	E_NORMAL_CAM_HANDLER_SEQ_STEPS.COUPLER_DETECT_IMAGE_ACQUIRE:
		gotoNextStep(gigECameraHandler.oImageAcquired, E_NORMAL_CAM_HANDLER_SEQ_STEPS.COUPLER_DETECT_IMAGE_PROCESSING);
		gotoNextStep(gigECameraHandler.oError, E_NORMAL_CAM_HANDLER_SEQ_STEPS.COUPLER_DETECT_FAILED);
	
	E_NORMAL_CAM_HANDLER_SEQ_STEPS.COUPLER_DETECT_IMAGE_PROCESSING:
		iCouplerProcessor.ic_process(iRawImage := rawImageCopy, iProcessedImage := processedImage, iDisplayableImage := displayableProcessedImage);
		gotoNextStep(iCouplerProcessor.ic_processingReady(), E_NORMAL_CAM_HANDLER_SEQ_STEPS.COUPLER_DETECT_DONE);
		gotoNextStep(iCouplerProcessor.ic_processingError(), E_NORMAL_CAM_HANDLER_SEQ_STEPS.COUPLER_DETECT_FAILED);

	E_NORMAL_CAM_HANDLER_SEQ_STEPS.COUPLER_DETECT_DONE:
		gotoNextStep(NOT iDetectCoupler, E_NORMAL_CAM_HANDLER_SEQ_STEPS.INIT);
	
	E_NORMAL_CAM_HANDLER_SEQ_STEPS.COUPLER_DETECT_FAILED:
		gotoNextStep(NOT iDetectCoupler, E_NORMAL_CAM_HANDLER_SEQ_STEPS.INIT);

// --------------------------------- MIRROR DETECT
	E_NORMAL_CAM_HANDLER_SEQ_STEPS.MIRROR_DETECT_ENABLE_LIGHT:
		gotoNextStep(isTimeExpired(T#500MS), E_NORMAL_CAM_HANDLER_SEQ_STEPS.MIRROR_DETECT_IMAGE_ACQUIRE);

	E_NORMAL_CAM_HANDLER_SEQ_STEPS.MIRROR_DETECT_IMAGE_ACQUIRE:
		gotoNextStep(gigECameraHandler.oImageAcquired, E_NORMAL_CAM_HANDLER_SEQ_STEPS.MIRROR_DETECT_IMAGE_PROCESSING);
		gotoNextStep(gigECameraHandler.oError, E_NORMAL_CAM_HANDLER_SEQ_STEPS.MIRROR_DETECT_FAILED);
	
	E_NORMAL_CAM_HANDLER_SEQ_STEPS.MIRROR_DETECT_IMAGE_PROCESSING:
		iMirrorProcessor.ic_process(iRawImage := rawImageCopy, iProcessedImage := processedImage, iDisplayableImage := displayableProcessedImage, iCameraPtr := gigECameraHandler.oCameraPtr, iCouplerCenterPoint := iCouplerProcessor.ic_getCenterPoint());
		gotoNextStep(iMirrorProcessor.ic_processingReady(), E_NORMAL_CAM_HANDLER_SEQ_STEPS.MIRROR_DETECT_DONE);
		gotoNextStep(iMirrorProcessor.ic_processingError(), E_NORMAL_CAM_HANDLER_SEQ_STEPS.MIRROR_DETECT_FAILED);

	E_NORMAL_CAM_HANDLER_SEQ_STEPS.MIRROR_DETECT_DONE:
		gotoNextStep(NOT iDetectMirror, E_NORMAL_CAM_HANDLER_SEQ_STEPS.INIT);
	
	E_NORMAL_CAM_HANDLER_SEQ_STEPS.MIRROR_DETECT_FAILED:
		gotoNextStep(NOT iDetectMirror, E_NORMAL_CAM_HANDLER_SEQ_STEPS.INIT);

ELSE
	step := E_NORMAL_CAM_HANDLER_SEQ_STEPS.INIT;
END_CASE
callMeRightAfterSwitchCase(TRUE, IING.STRING_BLANK);



gigECameraHandler(
	iDoIt := (step = E_NORMAL_CAM_HANDLER_SEQ_STEPS.UNDER_LIGHT_TEST_IMAGE_ACQUIRE),
	iReset := reset
);



oUnderlightOn := stepInBetween(E_NORMAL_CAM_HANDLER_SEQ_STEPS.UNDER_LIGHT_TEST_ENABLE_LIGHT, E_NORMAL_CAM_HANDLER_SEQ_STEPS.UNDER_LIGHT_TEST_IMAGE_PROCESSING)
	OR stepInBetween(E_NORMAL_CAM_HANDLER_SEQ_STEPS.COUPLER_DETECT_ENABLE_LIGHT, E_NORMAL_CAM_HANDLER_SEQ_STEPS.COUPLER_DETECT_IMAGE_PROCESSING);

oLaserLightOn := stepInBetween(E_NORMAL_CAM_HANDLER_SEQ_STEPS.LASER_LIGHT_TEST_ENABLE_LIGHT, E_NORMAL_CAM_HANDLER_SEQ_STEPS.LASER_LIGHT_TEST_IMAGE_PROCESSING);
//	OR 

oUnderLightTestOk := (step = E_NORMAL_CAM_HANDLER_SEQ_STEPS.UNDER_LIGHT_TEST_OK);
oUnderLightTestFailed := (step = E_NORMAL_CAM_HANDLER_SEQ_STEPS.UNDER_LIGHT_TEST_FAILED);

oLaserLightTestOk := (step = E_NORMAL_CAM_HANDLER_SEQ_STEPS.LASER_LIGHT_TEST_OK);
oLaserLightTestFailed := (step = E_NORMAL_CAM_HANDLER_SEQ_STEPS.LASER_LIGHT_TEST_FAILED);

oCouplerDetectDone := (step = E_NORMAL_CAM_HANDLER_SEQ_STEPS.COUPLER_DETECT_DONE);

oCouplerDetectFailed := (step = E_NORMAL_CAM_HANDLER_SEQ_STEPS.COUPLER_DETECT_FAILED);


mHmi();

METHOD PRIVATE mHmi
END_METHOD

METHOD PUBLIC stepAsString : T_SHORT_STR
stepAsString := TO_STRING(step);
END_METHOD

END_FUNCTION_BLOCK

// ---- POUs/HP/CURING_STATION/VISION/FB_GigECamHandler.TcPOU
FUNCTION_BLOCK FB_GigECamHandler EXTENDS FB_StepperProgram	// Wrapper/handler for gigE cameras, handles camera resetting, then images can be acquired (and converted)
VAR_INPUT
	iDoIt:						BOOL;		// 
	iDoConversion:				BOOL;
	iColorSpaceTransform:		ETcVnColorSpaceTransform;
	iReset:						BOOL;
END_VAR
VAR_OUTPUT
	oReadyForOperation:		BOOL;
	oImageAcquired:			BOOL;
	oDone:					BOOL;
	oError:					BOOL;
	
	oRawImage:				ITcVnImage;
	oConvertedImage:		ITcVnImage;
	
	oCameraPtr:				POINTER TO FB_VN_GevCameraControl;
	oScalingFactor:			LREAL;
END_VAR
VAR_IN_OUT
END_VAR
VAR
	step:					E_GIGE_CAM_HANDLER_SEQ_STEPS;
	hResult:				HRESULT;
	visionState:			ETcVnCameraState;
	visionStateError:		BOOL;
	ioCameraFb:				FB_VN_GevCameraControl;
	
	
END_VAR


visionState := ioCameraFb.GetState();
visionStateError := (visionState = TCVN_CS_ERROR);



callMeRightBeforeSwitchCase(ADR(step));
CASE step OF
	E_GIGE_CAM_HANDLER_SEQ_STEPS.INIT:
		gotoNextStep(iReset OR iDoIt AND (visionState = TCVN_CS_ERROR), E_GIGE_CAM_HANDLER_SEQ_STEPS.RESET_CAMERA);
		gotoNextStep(iReset OR iDoIt AND (visionState = TCVN_CS_INITIAL), E_GIGE_CAM_HANDLER_SEQ_STEPS.READY_FOR_OPERATION);

	E_GIGE_CAM_HANDLER_SEQ_STEPS.RESET_CAMERA:
		hResult := ioCameraFb.Reset();
		hResult := FC_GetCameraScalingFactor(iCameraPtr := oCameraPtr, iHrPrev := hResult, ioScale := oScalingFactor);
		
		gotoNextStep(hResult = S_OK, E_GIGE_CAM_HANDLER_SEQ_STEPS.READY_FOR_OPERATION);
		gotoNextStep(hResult = S_FALSE, E_GIGE_CAM_HANDLER_SEQ_STEPS.ERROR);
	
	E_GIGE_CAM_HANDLER_SEQ_STEPS.READY_FOR_OPERATION:
		gotoNextStep(iDoIt, E_GIGE_CAM_HANDLER_SEQ_STEPS.TRIGGER_CAMERA);
	
	E_GIGE_CAM_HANDLER_SEQ_STEPS.TRIGGER_CAMERA:
		hResult := ioCameraFb.TriggerImage();
		gotoNextStep(FAILED(hResult) OR visionStateError, E_GIGE_CAM_HANDLER_SEQ_STEPS.ERROR);
		gotoNextStep(SUCCEEDED(hresult) AND (visionState = TCVN_CS_STARTACQUISITION) , E_GIGE_CAM_HANDLER_SEQ_STEPS.START_ACQUISITION);
	
	E_GIGE_CAM_HANDLER_SEQ_STEPS.START_ACQUISITION:
		hResult := ioCameraFb.StartAcquisition();
		gotoNextStep(FAILED(hResult) OR visionStateError, E_GIGE_CAM_HANDLER_SEQ_STEPS.ERROR);
		gotoNextStep(SUCCEEDED(hresult) AND (visionState = TCVN_CS_ACQUIRING) , E_GIGE_CAM_HANDLER_SEQ_STEPS.ACQUIRING);
		
	E_GIGE_CAM_HANDLER_SEQ_STEPS.ACQUIRING:
		hResult := ioCameraFb.GetCurrentImageUndistorted(oRawImage);
		gotoNextStep(iDoConversion AND SUCCEEDED(hResult) AND (oRawImage <> IING.ZERO_POINTER), E_GIGE_CAM_HANDLER_SEQ_STEPS.DO_COLOR_CONVERSION);
		gotoNextStep(NOT iDoConversion AND SUCCEEDED(hResult) AND (oRawImage <> IING.ZERO_POINTER), E_GIGE_CAM_HANDLER_SEQ_STEPS.ACQUIRED);
		
		gotoNextStep(FAILED(hResult), E_GIGE_CAM_HANDLER_SEQ_STEPS.ERROR); 
			
	E_GIGE_CAM_HANDLER_SEQ_STEPS.DO_COLOR_CONVERSION:
		hResult := F_VN_ConvertColorSpace(ipSrcImage := oRawImage, ipDestImage := oConvertedImage, eTransform := iColorSpaceTransform, hrPrev:= hResult);
		gotoNextStep(SUCCEEDED(hResult), E_GIGE_CAM_HANDLER_SEQ_STEPS.ACQUIRED);
		gotoNextStep(FAILED(hResult), E_GIGE_CAM_HANDLER_SEQ_STEPS.ERROR);
	
	E_GIGE_CAM_HANDLER_SEQ_STEPS.ACQUIRED:
		gotoNextStep(NOT iDoIt, E_GIGE_CAM_HANDLER_SEQ_STEPS.INIT);
	
	
	E_GIGE_CAM_HANDLER_SEQ_STEPS.ERROR:
		gotoNextStep(iReset, E_GIGE_CAM_HANDLER_SEQ_STEPS.INIT);
		
	
	
ELSE
	step := E_GIGE_CAM_HANDLER_SEQ_STEPS.INIT;
END_CASE
callMeRightAfterSwitchCase(TRUE, IING.STRING_BLANK);

oCameraPtr := adr(ioCameraFb);


oReadyForOperation := (step = E_GIGE_CAM_HANDLER_SEQ_STEPS.READY_FOR_OPERATION);
oImageAcquired := (step = E_GIGE_CAM_HANDLER_SEQ_STEPS.ACQUIRING);
oError := (step = E_GIGE_CAM_HANDLER_SEQ_STEPS.ERROR);
oDone := (step = E_GIGE_CAM_HANDLER_SEQ_STEPS.DONE);

METHOD PRIVATE calcScaleFactor : LREAL
END_METHOD

END_FUNCTION_BLOCK

// ---- POUs/HP/CURING_STATION/VISION/Mirror/FC_GetCameraScalingFactor.TcPOU
FUNCTION FC_GetCameraScalingFactor : HRESULT
VAR_INPUT
	iCameraPtr:		POINTER TO FB_VN_GevCameraControl;
	iHrPrev:			HRESULT;
END_VAR
VAR_IN_OUT
	ioScale:		LREAL;		// Will contain the millimeters for ONE pixel = scale
END_VAR
VAR
 	cameraMatrix:				TcVnMatrix3x3_LREAL;
    distortionCoefficients:		TcVnArray8_LREAL;
    rotationMatrix:				TcVnMatrix3x3_LREAL;
    translationVector:			TcVnVector3_LREAL;
	//hResult:					HRESULT;
	singlePixelPoint1:			TcVnPoint2_REAL := [0, 0];
	singlePixelPoint2:			TcVnPoint2_REAL := [0, 1];
END_VAR
VAR CONSTANT

END_VAR

// Get camera calibration parameters
iCameraPtr^.GetCameraMatrix(aCameraMatrix := cameraMatrix);
iCameraPtr^.GetDistortionCoefficients(aDistortionCoefficients := distortionCoefficients);
iCameraPtr^.GetRotationMatrix(aRotationMatrix := rotationMatrix);
iCameraPtr^.GetTranslationVector(aTranslationVector := translationVector);

singlePixelPoint1[VISION.X_COORD] := 0;
singlePixelPoint1[VISION.Y_COORD] := 0;

singlePixelPoint2[VISION.X_COORD] := 0;
singlePixelPoint2[VISION.Y_COORD] := 1;


// We ask to give the distance of point1 to point2 = 1 pixel -> this will give us the scaling factor
FC_GetCameraScalingFactor := F_VN_ImagePointsWorldDistance( 
	aImagePoint1 :=				singlePixelPoint1,
	aImagePoint2 :=				singlePixelPoint2,
	fWorldDistance :=			ioScale,
	aCameraMatrix :=			cameraMatrix,
	aDistortionCoefficients :=	distortionCoefficients,
	aRotationMatrix :=			rotationMatrix,
	aTranslationVector :=		translationVector,
	fZ :=						0,
	hrPrev :=					iHrPrev
);

END_FUNCTION

// ---- POUs/HP/CURING_STATION/VISION/Coupler/FB_CouplerImageProcessor.TcPOU
FUNCTION_BLOCK FB_CouplerImageProcessor	EXTENDS FB_StepperProgram IMPLEMENTS I_ImageProcessor		// FB responsible for VISION program detecting the coupler
VAR
	step:						E_COUPLER_PROCESSOR_STEPS;
	hResult:					HRESULT;

	rightEdgeStartPoint:		TcVnPoint2_REAL;
	rightEdgeEndPoint:			TcVnPoint2_REAL;
	rightEdgeResultContainer:	ITcVnContainer;	

	rightEdgePoint:				TcVnPoint2_REAL;
	topEdgePoints:				ARRAY [0..5] OF TcVnPoint2_REAL;
	bottomEdgePoints:			ARRAY [0..5] OF TcVnPoint2_REAL;

	topEdgestartPoint:			TcVnPoint2_REAL;
	topEdgeEndPoint:			TcVnPoint2_REAL;
	topEdgeEdgeResultContainer:	ITcVnContainer;	

	startPoint3:				TcVnPoint2_REAL;
	endPoint3:					TcVnPoint2_REAL;
	bottomEdgeResultContainer:	ITcVnContainer;
	
	i:							ULINT;

	topEdgePointAverage:		TcVnPoint2_REAL;
	bottomEdgePointAverage:		TcVnPoint2_REAL;
	
	// Result of the vision operation
	centerpoint:				TcVnPoint2_REAL;


	// Set throug hinterfaces
	doProcessing:				BOOL;
	rawImage:					ITcVnImage;				// Not owned, do not clear
	processedImage:				ITcVnImage;				// NOT owned, DO NOT clear
	displayableProcessedImage:	ITcVnDisplayableImage;	// Not owned, do not clear
	
	// 'Constants'
	searchLines:				UDINT;
	minIntensityDiff:			REAL;
	searchToLeftXOffset:		REAL;
END_VAR
VAR_STAT PERSISTENT
	settings:	ST_COUPLER_DETECT_SETTINGS;
END_VAR

searchLines := 5;
minIntensityDiff := 45;
searchToLeftXOffset := 40;

callMeRightBeforeSwitchCase(ADR(step));
CASE step OF
	E_COUPLER_PROCESSOR_STEPS.INIT:
		gotoNextStep(doProcessing, E_COUPLER_PROCESSOR_STEPS.LOCATE_RIGHT_EDGE);

	E_COUPLER_PROCESSOR_STEPS.LOCATE_RIGHT_EDGE:
		//mInternalCleanup();
		rightEdgeStartPoint[VISION.X_COORD] :=		1000;
		rightEdgeStartPoint[VISION.Y_COORD] :=		1000;
		rightEdgeEndPoint[VISION.X_COORD] :=		550;
		rightEdgeEndPoint[VISION.Y_COORD] :=		1000;

		hResult := F_VN_LocateEdge(
			ipSrcImage :=		rawImage, 
			ipEdgePoints :=		rightEdgeResultContainer, 
			aStartPoint :=		rightEdgeStartPoint, 
			aEndPoint :=		rightEdgeEndPoint, 
			eEdgeDirection :=	ETcVnEdgeDirection.TCVN_ED_Light_TO_Dark, 
			fMinStrength :=		minIntensityDiff, 
			nSearchLines :=		searchLines, 				// Was 5!?!?!
			hrPrev :=			hResult
		);
		// Reads the result from the container and stores to the rightEdgePoint -> Used in the next operations for calculating an offset
//		hResult := F_VN_GetAt_TcVnVector2_REAL(ipContainer := rightEdgeResultContainer, aElement := rightEdgePoint, nIndex := 0, hrPrev := hResult);		// ONLY 1 point USED!!
		hResult := FC_ExtractFromContainerAndCalculateAvg(ipContainer := rightEdgeResultContainer, iNumOfElements := (searchLines - 1), hrPrev := hResult, ioResult := rightEdgePoint);	


		gotoNextStep(SUCCEEDED(hResult), E_COUPLER_PROCESSOR_STEPS.LOCATE_TOP_EDGE);
		gotoNextStep(FAILED(hResult), E_COUPLER_PROCESSOR_STEPS.ERROR);
	
	E_COUPLER_PROCESSOR_STEPS.LOCATE_TOP_EDGE:
		topEdgestartPoint[VISION.X_COORD] :=	rightEdgePoint[VISION.X_COORD] - searchToLeftXOffset;
		topEdgestartPoint[VISION.Y_COORD] :=	600;
		topEdgeEndPoint[VISION.X_COORD] :=		rightEdgePoint[VISION.X_COORD] - searchToLeftXOffset;
		topEdgeEndPoint[VISION.Y_COORD] :=		1000;	
		
		hResult := F_VN_LocateEdge(
			ipSrcImage :=		rawImage,
			ipEdgePoints :=		topEdgeEdgeResultContainer,
			aStartPoint :=		topEdgestartPoint,
			aEndPoint :=		topEdgeEndPoint,
			eEdgeDirection :=	ETcVnEdgeDirection.TCVN_ED_Light_TO_Dark,
			fMinStrength :=		minIntensityDiff,
			nSearchLines :=		searchLines,		// Was 4!?!?!
			hrPrev :=			hResult, 
		);
		gotoNextStep(SUCCEEDED(hResult), E_COUPLER_PROCESSOR_STEPS.LOCATE_BOTTOM_EDGE);
		gotoNextStep(FAILED(hResult), E_COUPLER_PROCESSOR_STEPS.ERROR);

	E_COUPLER_PROCESSOR_STEPS.LOCATE_BOTTOM_EDGE:
		startPoint3[VISION.X_COORD] :=		rightEdgePoint[0] - searchToLeftXOffset;
		startPoint3[VISION.Y_COORD] :=		1400;
		endPoint3[VISION.X_COORD] :=		rightEdgePoint[0] - searchToLeftXOffset;
		endPoint3[VISION.Y_COORD] :=		1000;	

		hResult := F_VN_LocateEdge(
			ipSrcImage :=		rawImage,
			ipEdgePoints :=		bottomEdgeResultContainer,
			aStartPoint :=		startPoint3,
			aEndPoint :=		endPoint3,
			eEdgeDirection :=	ETcVnEdgeDirection.TCVN_ED_Light_TO_Dark,
			fMinStrength :=		minIntensityDiff,
			nSearchLines :=		searchLines,				// Was 4!?!?!
			hrPrev :=			hResult 
		);
		gotoNextStep(SUCCEEDED(hResult), E_COUPLER_PROCESSOR_STEPS.DRAW_POINTS);
		gotoNextStep(FAILED(hResult), E_COUPLER_PROCESSOR_STEPS.ERROR);

	E_COUPLER_PROCESSOR_STEPS.DRAW_POINTS:
		hResult := F_VN_DrawPoints(ipPoints := rightEdgeResultContainer, ipDestImage := processedImage, eShape := ETcVnDrawShape.TCVN_DS_X, aColor := Color.Lime, hrPrev := hResult);
		hResult := F_VN_DrawPoints(ipPoints := topEdgeEdgeResultContainer, ipDestImage := processedImage, eShape := ETcVnDrawShape.TCVN_DS_X, aColor := Color.Lime, hrPrev := hResult);
		hResult := F_VN_DrawPoints(ipPoints := bottomEdgeResultContainer, ipDestImage := processedImage, eShape := ETcVnDrawShape.TCVN_DS_X, aColor := Color.Lime, hrPrev := hResult);

		hResult := FC_ExtractFromContainerAndCalculateAvg(ipContainer := topEdgeEdgeResultContainer, iNumOfElements := (searchLines - 1), hrPrev := hResult, ioResult := topEdgePointAverage);
		hResult := FC_ExtractFromContainerAndCalculateAvg(ipContainer := bottomEdgeResultContainer, iNumOfElements := (searchLines - 1), hrPrev := hResult, ioResult := bottomEdgePointAverage);
		centerpoint := FC_CalculateCenterPoint(topEdgePointAverage, bottomEdgePointAverage);

		gotoNextStep(SUCCEEDED(hResult), E_COUPLER_PROCESSOR_STEPS.MAKE_DISPLAYABLE);
		gotoNextStep(FAILED(hResult), E_COUPLER_PROCESSOR_STEPS.ERROR);	

	E_COUPLER_PROCESSOR_STEPS.MAKE_DISPLAYABLE:
		hResult := F_VN_CopyIntoDisplayableImage(processedImage, displayableProcessedImage, hResult);
		gotoNextStep(SUCCEEDED(hResult), E_COUPLER_PROCESSOR_STEPS.DONE);
		gotoNextStep(FAILED(hResult), E_COUPLER_PROCESSOR_STEPS.ERROR);
	
	E_COUPLER_PROCESSOR_STEPS.DONE:
		gotoNextStep(NOT doProcessing, E_COUPLER_PROCESSOR_STEPS.INIT);
	
	E_COUPLER_PROCESSOR_STEPS.ERROR:
		gotoNextStep(NOT doProcessing, E_COUPLER_PROCESSOR_STEPS.INIT);
	
ELSE
	step := E_COUPLER_PROCESSOR_STEPS.INIT;
END_CASE
callMeRightAfterSwitchCase(TRUE, IING.STRING_BLANK);

METHOD PRIVATE _mInternalCleanup
doProcessing := FALSE;
END_METHOD

METHOD ic_cancelProcessing
VAR_INPUT
END_VAR
doProcessing := FALSE;
END_METHOD

METHOD ic_getCenterPoint : TcVnPoint2_REAL
ic_getCenterPoint := centerpoint;
END_METHOD

METHOD ic_process
VAR_INPUT
	iRawImage:			ITcVnImage;
	iProcessedImage:	ITcVnImage;
	iDisplayableImage:	ITcVnDisplayableImage;
END_VAR
doProcessing := TRUE;
rawImage := iRawImage;
processedImage := iProcessedImage;
displayableProcessedImage := iDisplayableImage;
END_METHOD

METHOD public ic_processingError : BOOL
ic_processingError := (step = E_COUPLER_PROCESSOR_STEPS.ERROR);
END_METHOD

METHOD public ic_processingReady : BOOL
ic_processingReady := (step = E_COUPLER_PROCESSOR_STEPS.DONE);
END_METHOD

METHOD PUBLIC stepAsString : T_SHORT_STR
stepAsString := TO_STRING(step);
END_METHOD

END_FUNCTION_BLOCK

// ---- POUs/HP/CURING_STATION/VISION/HelperFunctions/FC_ExtractFromContainerAndCalculateAvg.TcPOU
FUNCTION FC_ExtractFromContainerAndCalculateAvg  : HRESULT		// Calculates average X and Y of the search result stored in container
VAR_INPUT
	ipContainer:	ITcVnContainer;
	iNumOfElements:	UDINT;
	hrPrev	:	HRESULT;	(* HRESULT indicating the result of previous operations (If SUCCEEDED(hrPrev) equals false, no operation is executed.) *)
END_VAR
VAR_IN_OUT
	ioResult:		TcVnPoint2_REAL;
END_VAR
VAR
	i:				UDINT;
	helperPoint:			TcVnPoint2_REAL;
	hResult:		HRESULT;
END_VAR

ioResult[VISION.X_COORD] := 0;
ioResult[VISION.Y_COORD] := 0;
hResult := hrPrev;

// Fetches result and stores to element
FOR i := 0 TO (iNumOfElements - 1) DO
	hResult := F_VN_GetAt_TcVnVector2_REAL(ipContainer := ipContainer, aElement := helperPoint, nIndex := i, hrPrev := hResult);

	// Accumulate all X's and all Y's
	ioResult[VISION.X_COORD] := ioResult[VISION.X_COORD] + helperPoint[VISION.X_COORD];
	ioResult[VISION.Y_COORD] := ioResult[VISION.Y_COORD] + helperPoint[VISION.Y_COORD];
END_FOR

// Averages the X and Y's
ioResult[VISION.X_COORD] := ioResult[VISION.X_COORD] / UDINT_TO_REAL(iNumOfElements);
ioResult[VISION.Y_COORD] := ioResult[VISION.Y_COORD] / UDINT_TO_REAL(iNumOfElements);

FC_ExtractFromContainerAndCalculateAvg := hResult;

END_FUNCTION

// ---- POUs/HP/CURING_STATION/VISION/HelperFunctions/FC_CalculateCenterPoint.TcPOU
FUNCTION FC_CalculateCenterPoint : TcVnPoint2_REAL		// Calculates the center point (X and Y) of 2 points
VAR_INPUT
	iPoint1:		TcVnPoint2_REAL;
	iPoint2:		TcVnPoint2_REAL;
END_VAR

FC_CalculateCenterPoint[VISION.X_COORD] := (iPoint1[VISION.X_COORD] + iPoint2[VISION.X_COORD]) / 2;
FC_CalculateCenterPoint[VISION.Y_COORD] := (iPoint1[VISION.Y_COORD] + iPoint2[VISION.Y_COORD]) / 2;

END_FUNCTION

// ---- POUs/HP/CURING_STATION/VISION/GenericCameraHandler/FB_GenericCameraHandler.TcPOU
FUNCTION_BLOCK FB_GenericCameraHandler EXTENDS FB_StepperProgram	
VAR_INPUT
	iDoUnderLightTest:		BOOL;
	iDoLaserTest:			BOOL;
	iDetectCoupler:			BOOL;
	iDetectMirror:			BOOL;
	
	iCouplerProcessor:		I_ImageProcessor;		// FB implementing
	iMirrorProcessor:		I_ImageProcessor;
	
END_VAR
VAR_OUTPUT
	oUnderLightTestOk:			BOOL;
	oUnderLightTestFailed:		BOOL;
	oLaserLightTestOk:			BOOL;
	oLaserLightTestFailed:		BOOL;

	oCouplerDetectDone:			BOOL;
	oCouplerDetectFailed:		BOOL;

	oHmi:						ST_NORMAL_CAM_HANDLER_HMI;
	
	oUnderlightOn:				BOOL;
	oLaserLightOn:				BOOL;
END_VAR
VAR_IN_OUT
END_VAR
VAR
	step:					E_NORMAL_CAM_HANDLER_SEQ_STEPS;
	service:				ST_NORMAL_CAM_HANDLER_SERVICE;
	
	visionState:			ETcVnCameraState;
	gigECameraHandler:		FB_GigECamHandler;
	hResult:				HRESULT;
	
	rectangleArea:			TcVnRectangle_UDINT;
	rawImageCopy:			ITcVnImage;				// Image of either under light/laser
	processedImage:			ITcVnImage;
	displayableProcessedImage:	ITcVnDisplayableImage;

	averagePixelValue:		TcVnVector4_LREAL;
	
	reset:					BOOL;
	

END_VAR
VAR PERSISTENT
	settings:				ST_NORMAL_CAM_HANDLER_SETTINGS;
END_VAR

reset := iControlSignals.resetPulse;



callMeRightBeforeSwitchCase(ADR(step));
CASE step OF
	E_NORMAL_CAM_HANDLER_SEQ_STEPS.INIT:
		gotoNextStep(iDoUnderLightTest OR service.doUnderLightTest, E_NORMAL_CAM_HANDLER_SEQ_STEPS.UNDER_LIGHT_TEST_ENABLE_LIGHT);
		gotoNextStep(iDoLaserTest OR service.doLaserTest, E_NORMAL_CAM_HANDLER_SEQ_STEPS.LASER_LIGHT_TEST_ENABLE_LIGHT);
		gotoNextStep(iDetectCoupler, E_NORMAL_CAM_HANDLER_SEQ_STEPS.COUPLER_DETECT_ENABLE_LIGHT);
		gotoNextStep(iDetectMirror, E_NORMAL_CAM_HANDLER_SEQ_STEPS.MIRROR_DETECT_ENABLE_LIGHT);



// --------------------------------- COUPLER DETECT
	E_NORMAL_CAM_HANDLER_SEQ_STEPS.COUPLER_DETECT_ENABLE_LIGHT:
		gotoNextStep(isTimeExpired(T#500MS), E_NORMAL_CAM_HANDLER_SEQ_STEPS.COUPLER_DETECT_IMAGE_ACQUIRE);

	E_NORMAL_CAM_HANDLER_SEQ_STEPS.COUPLER_DETECT_IMAGE_ACQUIRE:
		gotoNextStep(gigECameraHandler.oImageAcquired, E_NORMAL_CAM_HANDLER_SEQ_STEPS.COUPLER_DETECT_IMAGE_PROCESSING);
		gotoNextStep(gigECameraHandler.oError, E_NORMAL_CAM_HANDLER_SEQ_STEPS.COUPLER_DETECT_FAILED);
	
	E_NORMAL_CAM_HANDLER_SEQ_STEPS.COUPLER_DETECT_IMAGE_PROCESSING:
		iCouplerProcessor.ic_process(iRawImage := rawImageCopy, iProcessedImage := processedImage, iDisplayableImage := displayableProcessedImage);
		gotoNextStep(iCouplerProcessor.ic_processingReady(), E_NORMAL_CAM_HANDLER_SEQ_STEPS.COUPLER_DETECT_DONE);
		gotoNextStep(iCouplerProcessor.ic_processingError(), E_NORMAL_CAM_HANDLER_SEQ_STEPS.COUPLER_DETECT_FAILED);

	E_NORMAL_CAM_HANDLER_SEQ_STEPS.COUPLER_DETECT_DONE:
		gotoNextStep(NOT iDetectCoupler, E_NORMAL_CAM_HANDLER_SEQ_STEPS.INIT);
	
	E_NORMAL_CAM_HANDLER_SEQ_STEPS.COUPLER_DETECT_FAILED:
		gotoNextStep(NOT iDetectCoupler, E_NORMAL_CAM_HANDLER_SEQ_STEPS.INIT);


ELSE
	step := E_NORMAL_CAM_HANDLER_SEQ_STEPS.INIT;
END_CASE
callMeRightAfterSwitchCase(TRUE, IING.STRING_BLANK);



gigECameraHandler(
	iDoIt := (step = E_NORMAL_CAM_HANDLER_SEQ_STEPS.UNDER_LIGHT_TEST_IMAGE_ACQUIRE),
	iReset := reset
);



oUnderlightOn := stepInBetween(E_NORMAL_CAM_HANDLER_SEQ_STEPS.UNDER_LIGHT_TEST_ENABLE_LIGHT, E_NORMAL_CAM_HANDLER_SEQ_STEPS.UNDER_LIGHT_TEST_IMAGE_PROCESSING)
	OR stepInBetween(E_NORMAL_CAM_HANDLER_SEQ_STEPS.COUPLER_DETECT_ENABLE_LIGHT, E_NORMAL_CAM_HANDLER_SEQ_STEPS.COUPLER_DETECT_IMAGE_PROCESSING);

oLaserLightOn := stepInBetween(E_NORMAL_CAM_HANDLER_SEQ_STEPS.LASER_LIGHT_TEST_ENABLE_LIGHT, E_NORMAL_CAM_HANDLER_SEQ_STEPS.LASER_LIGHT_TEST_IMAGE_PROCESSING);
//	OR 

oUnderLightTestOk := (step = E_NORMAL_CAM_HANDLER_SEQ_STEPS.UNDER_LIGHT_TEST_OK);
oUnderLightTestFailed := (step = E_NORMAL_CAM_HANDLER_SEQ_STEPS.UNDER_LIGHT_TEST_FAILED);

oLaserLightTestOk := (step = E_NORMAL_CAM_HANDLER_SEQ_STEPS.LASER_LIGHT_TEST_OK);
oLaserLightTestFailed := (step = E_NORMAL_CAM_HANDLER_SEQ_STEPS.LASER_LIGHT_TEST_FAILED);

oCouplerDetectDone := (step = E_NORMAL_CAM_HANDLER_SEQ_STEPS.COUPLER_DETECT_DONE);

oCouplerDetectFailed := (step = E_NORMAL_CAM_HANDLER_SEQ_STEPS.COUPLER_DETECT_FAILED);


mHmi();

METHOD PRIVATE mHmi
END_METHOD

METHOD PUBLIC stepAsString : T_SHORT_STR
stepAsString := TO_STRING(step);
END_METHOD

END_FUNCTION_BLOCK

// ---- POUs/HP/CURING_STATION/VISION/Mirror/FB_MirrorImageProcessor.TcPOU
FUNCTION_BLOCK FB_MirrorImageProcessor	EXTENDS FB_StepperProgram IMPLEMENTS I_MirrorImageProcessor		// FB responsible for VISION program detecting the mirror
VAR_INPUT
	iRecipes:					REFERENCE TO ST_Recipes;
END_VAR
VAR
	step:						E_MIRROR_PROCESSOR_STEPS;
	hResult:					HRESULT;
 
	cameraScale:				LREAL;		// 1 pixel in millimeters
	mirrorCenterToWeightCenterYDiffInPixels:	LREAL;
	mirrorHalfHeightInMm:			LREAL;

	upperEdgeStartPoint:		TcVnPoint2_REAL;
	upperEdgeEndPoint:			TcVnPoint2_REAL;
	upperEdgeResultContainer:	ITcVnContainer;	

	lowerEdgeStartPoint:		TcVnPoint2_REAL;
	lowerEdgeEndPoint:			TcVnPoint2_REAL;
	lowerEdgeResultContainer:	ITcVnContainer;	

	upperEdgePointAverage:		TcVnPoint2_REAL;
	lowerEdgePointAverage:		TcVnPoint2_REAL;

	mirrorCenterY:				REAL;
	// Result of the vision operation
	yOffsetInMm:					REAL;


	// Set through hinterfaces
	doProcessing:				BOOL;
	rawImage:					ITcVnImage;				// Not owned, do not clear
	processedImage:				ITcVnImage;				// NOT owned, DO NOT clear
	displayableProcessedImage:	ITcVnDisplayableImage;	// Not owned, do not clear
	
	// 'Constants'
	searchLines:				UDINT;
	minIntensityDiff:			REAL;
	verticalSearchYOffsetInPixels:		REAL;
	cameraPtr:					POINTER TO FB_VN_GevCameraControl;
	couplerCenterPoint:			TcVnPoint2_REAL;
END_VAR
VAR_STAT PERSISTENT
	settings:	ST_MIRROR_DETECT_SETTINGS;
END_VAR
VAR CONSTANT
	SINGLE_PIXEL_POINT1:	TcVnPoint2_REAL := [0, 0];
	SINGLE_PIXEL_POINT2:	TcVnPoint2_REAL := [0, 1];
END_VAR

searchLines := 1;
minIntensityDiff := 45;
verticalsearchYOffsetInPixels := 100;


callMeRightBeforeSwitchCase(ADR(step));
CASE step OF
	E_MIRROR_PROCESSOR_STEPS.INIT:
		gotoNextStep(doProcessing, E_MIRROR_PROCESSOR_STEPS.CALC_CENTER_POINT_OFFSET);

	E_MIRROR_PROCESSOR_STEPS.CALC_CENTER_POINT_OFFSET:
		hResult := FC_GetCameraScalingFactor(iCameraPtr := cameraPtr, iHrPrev := hResult, ioScale := cameraScale);

		mirrorCenterToWeightCenterYDiffInPixels := iRecipes.Station1To5.rMirrorCenterOffsetToWeightCenterY / cameraScale; // calculates the distance in px of the mirror centerpoint to weight centerpoint. Is used to determine currect positioning of the mirror 
	
		mirrorHalfHeightInMm := iRecipes.Station1To5.rMirrorDimensions[VISION.Y_COORD] / 2;				// HOX!!!!!   To be done either for 1..5 or 6..10
	
		// Detection from center to upper edge
		upperEdgeStartPoint[VISION.X_COORD] := LREAL_TO_REAL(couplerCenterPoint[VISION.X_COORD] - ((iRecipes.Station1To5.rCouplerGroveDepth) / cameraScale) + (iRecipes.Station1To5.rMirrorGripPointOffsetToEdgeX / cameraScale)) ;
		upperEdgeStartPoint[VISION.Y_COORD] := couplerCenterPoint[VISION.Y_COORD]; // Coupler centerpoint based Y Startpoint
		upperEdgeEndPoint[VISION.X_COORD] := upperEdgeStartPoint[VISION.X_COORD];	// Copy of start = thus same X
		upperEdgeEndPoint[VISION.Y_COORD] := LREAL_TO_REAL(couplerCenterpoint[VISION.Y_COORD] - ((mirrorHalfHeightInMm - iRecipes.Station1To5.rMirrorCenterOffsetToWeightCenterY) / cameraScale) - verticalSearchYOffsetInPixels);

		// Detection from center to lower edge
		lowerEdgeStartPoint[VISION.X_COORD] := LREAL_TO_REAL(couplerCenterPoint[VISION.X_COORD] - ((iRecipes.Station1To5.rCouplerGroveDepth) / cameraScale) + (iRecipes.Station1To5.rMirrorGripPointOffsetToEdgeX / cameraScale));
		lowerEdgeStartPoint[VISION.Y_COORD] := couplerCenterPoint[VISION.Y_COORD];
		lowerEdgeEndPoint[VISION.X_COORD] := lowerEdgeStartPoint[VISION.X_COORD];	// Copy of start = thus same X
		lowerEdgeEndPoint[VISION.Y_COORD] := LREAL_TO_REAL(couplerCenterpoint[VISION.Y_COORD] + ((mirrorHalfHeightInMm - iRecipes.Station1To5.rMirrorCenterOffsetToWeightCenterY) / cameraScale) + verticalSearchYOffsetInPixels);

		gotoNextStep(SUCCEEDED(hResult), E_MIRROR_PROCESSOR_STEPS.FIND_UPPER_EDGE); 
		gotoNextStep(FAILED(hResult), E_MIRROR_PROCESSOR_STEPS.ERROR); 

	E_MIRROR_PROCESSOR_STEPS.FIND_UPPER_EDGE:
		hResult := F_VN_LocateEdge(
			ipSrcImage :=			rawImage,
			ipEdgePoints :=			upperEdgeResultContainer,
			aStartPoint :=			upperEdgeStartPoint,
			aEndPoint :=			upperEdgeEndPoint,
			eEdgeDirection :=		ETcVnEdgeDirection.TCVN_ED_DARK_TO_LIGHT,
			fMinStrength :=			minIntensityDiff,
			nSearchLines :=			searchLines,
			hrPrev :=				hResult
		);
		hResult := FC_ExtractFromContainerAndCalculateAvg(ipContainer := upperEdgeResultContainer, iNumOfElements := (searchLines - 1), hrPrev := hResult, ioResult := upperEdgePointAverage);

		gotoNextStep(SUCCEEDED(hResult), E_MIRROR_PROCESSOR_STEPS.FIND_LOWER_EDGE); 
		gotoNextStep(FAILED(hResult), E_MIRROR_PROCESSOR_STEPS.ERROR); 

	E_MIRROR_PROCESSOR_STEPS.FIND_LOWER_EDGE:
		hResult := F_VN_LocateEdge(
			ipSrcImage :=			rawImage,
			ipEdgePoints :=			lowerEdgeResultContainer,
			aStartPoint :=			lowerEdgeStartPoint,
			aEndPoint :=			lowerEdgeEndPoint,
			eEdgeDirection :=		ETcVnEdgeDirection.TCVN_ED_DARK_TO_LIGHT,
			fMinStrength :=			minIntensityDiff,
			nSearchLines :=			searchLines,
			hrPrev :=				hResult
		);
		gotoNextStep(SUCCEEDED(hResult), E_MIRROR_PROCESSOR_STEPS.FIND_LOWER_EDGE); 
		gotoNextStep(FAILED(hResult), E_MIRROR_PROCESSOR_STEPS.ERROR); 

	E_MIRROR_PROCESSOR_STEPS.DRAW_POINTS:
		hResult := F_VN_DrawPoints(ipPoints := upperEdgeResultContainer, ipDestImage := processedImage, eShape := ETcVnDrawShape.TCVN_DS_X, aColor := Color.Lime, hrPrev := hResult);
		hResult := F_VN_DrawPoints(ipPoints := lowerEdgeResultContainer, ipDestImage := processedImage, eShape := ETcVnDrawShape.TCVN_DS_X, aColor := Color.Lime, hrPrev := hResult);

		// Vision found the edges of the mirror = Mirror Center
		mirrorCenterY := FC_CalculateYCenterPoint(upperEdgePointAverage, lowerEdgePointAverage);

		yOffsetInMm := LREAL_TO_REAL((couplerCenterPoint[VISION.Y_COORD] - mirrorCenterY - mirrorCenterToWeightCenterYDiffInPixels) * cameraScale);

		gotoNextStep(SUCCEEDED(hResult), E_COUPLER_PROCESSOR_STEPS.MAKE_DISPLAYABLE);
		gotoNextStep(FAILED(hResult), E_COUPLER_PROCESSOR_STEPS.ERROR);	

	E_MIRROR_PROCESSOR_STEPS.MAKE_DISPLAYABLE:
		hResult := F_VN_CopyIntoDisplayableImage(processedImage, displayableProcessedImage, hResult);
		gotoNextStep(SUCCEEDED(hResult), E_COUPLER_PROCESSOR_STEPS.DONE);
		gotoNextStep(FAILED(hResult), E_COUPLER_PROCESSOR_STEPS.ERROR);

	E_MIRROR_PROCESSOR_STEPS.DONE:
		gotoNextStep(NOT doProcessing, E_MIRROR_PROCESSOR_STEPS.INIT);
	
	E_MIRROR_PROCESSOR_STEPS.ERROR:
		gotoNextStep(NOT doProcessing, E_COUPLER_PROCESSOR_STEPS.INIT);
	
ELSE
	step := E_MIRROR_PROCESSOR_STEPS.INIT;
END_CASE
callMeRightAfterSwitchCase(TRUE, IING.STRING_BLANK);

METHOD PRIVATE _mInternalCleanup
doProcessing := FALSE;
END_METHOD

ACTION documentation:
(**









*)
END_ACTION

METHOD ic_cancelProcessing
VAR_INPUT
END_VAR
doProcessing := FALSE;
END_METHOD

METHOD ic_getResult : REAL
ic_getResult := yOffsetInMm;
END_METHOD

METHOD ic_process
VAR_INPUT
	iRawImage:				ITcVnImage;
	iProcessedImage:		ITcVnImage;
	iDisplayableImage:		ITcVnDisplayableImage;
	iCameraPtr:				POINTER TO FB_VN_GevCameraControl;
	iCouplerCenterPoint:	TcVnPoint2_REAL;					// Basis for next vision operations
END_VAR
doProcessing := TRUE;
rawImage := iRawImage;
processedImage := iProcessedImage;
displayableProcessedImage := iDisplayableImage;
cameraPtr := iCameraPtr;
couplerCenterPoint := iCouplerCenterPoint;
END_METHOD

METHOD public ic_processingError : BOOL
ic_processingError := (step = E_MIRROR_PROCESSOR_STEPS.ERROR);
END_METHOD

METHOD public ic_processingReady : BOOL
ic_processingReady := (step = E_MIRROR_PROCESSOR_STEPS.DONE);
END_METHOD

METHOD PUBLIC stepAsString : T_SHORT_STR
stepAsString := TO_STRING(step);
END_METHOD

END_FUNCTION_BLOCK

// ---- POUs/Sts/Datalog/FB_Datalogger2.TcPOU
FUNCTION_BLOCK FB_Datalogger2
VAR_INPUT
    iScaledTemp            : INT;
    stMirrorData         : REFERENCE TO ST_Vis_Mirror;
	stLaserData			: REFERENCE TO ST_Vis_Laser;
    bEnable             : BOOL;        // Rising edge = add one log entry
    bSave               : BOOL;        // Rising edge = write CSV

    Stepperpos          : LREAL;
    SensorVal           : INT;
    StepperHomed        : BOOL;
    Var4                : BOOL;
    Var5                : LREAL;
    Var6                : INT;
    Var7                : LREAL;
    Var8                : BOOL;
    Var9                : BOOL;
    Error               : BOOL;

END_VAR

VAR_OUTPUT
    bBusy               : BOOL;
    bDone               : BOOL;
    bError              : BOOL;
	bArrayWriteDone		: BOOL;
END_VAR

VAR
    // Ring buffer
    aLog        : ARRAY[0..999] OF ST_LogEntry;
    WriteIndex  : UINT := 0;
    Count       : UINT := 0;
    ReadIndex   : UINT := 0;

    // Edge detectors
    rEnable     : R_TRIG;
    rSave       : R_TRIG;

    // File handling
    fbOpen      : FB_FileOpen;
    fbWrite     : FB_FileWrite;
    fbClose     : FB_FileClose;

    hFile       : UINT;
    sLine       : STRING(255);
    sFile       : STRING(255) := 'C:\ProgramData\Beckhoff\TwinCAT\3.1\Boot\datalog2.csv';
    sCRLF       : STRING(2) := '$R$L';

    bHeaderWritten : BOOL := FALSE;
    index          : UINT;

    // State machine
    eState     : INT := 0;

    // Time stamp
    fbSysTime  : FB_LocalSystemTime;
// 					sNetID :='192.168.1.11.1.1',
// 					bEnable := TRUE);
    CurrentDT  : DT;
	
	WriteDoneTof		: TOF;
	DoneTof				: TOF;
	bDoneStatus	: BOOL;
	bWriteDone	: BOOL;
	
END_VAR

WriteDoneTof( IN := bWriteDone	, PT := T#0.2S, Q => bArrayWriteDone);
DoneTof(IN := bDoneStatus, PT := T#0.2S, Q => bDone);
bWriteDone := FALSE;
bDoneStatus := FALSE;

//  GET SYSTEM TIMESTAMP

fbSysTime(sNetID :='192.168.1.11.1.1',
					bEnable := TRUE);
//CurrentDT :=  (fbSysTime.systemTime);


//  RISING EDGE OF bEnable 

rEnable(CLK := bEnable);

IF rEnable.Q AND NOT bBusy THEN

    aLog[WriteIndex].tStamp := fbSysTime.systemTime;
    aLog[WriteIndex].Var1   := stMirrorData.rMirrorOffsetToCalPoints[1];
    aLog[WriteIndex].Var2   := stLaserData.rLaserOffsetToSetPoint[0];
    aLog[WriteIndex].Var3   := iScaledTemp;

    // Advance write pointer
    WriteIndex := WriteIndex + 1;
	bWriteDone := TRUE;
    IF WriteIndex > 999 THEN WriteIndex := 0; END_IF

    // Increment count up to 1000
    IF Count < 1000 THEN Count := Count + 1; END_IF
END_IF


//    RISING EDGE OF bSave, START FILE WRITE SEQUENCE

rSave(CLK := bSave);

IF rSave.Q AND (Count > 0) AND (NOT bBusy) THEN
    bBusy  := TRUE;
    bError := FALSE;
    eState := 10;
END_IF



CASE eState OF


// Idle

0:
    // do nothing bdone:=false????????


//  OPEN FILE (APPEND MODE)

10:
    fbOpen(
        sPathName := sFile,
        nMode     := FOPEN_MODEAPPEND,
        ePath     := PATH_GENERIC,
        bExecute  := TRUE
    );
    eState := 20;


// WAIT OPEN

20:
    fbOpen(bExecute := FALSE);

    IF NOT fbOpen.bBusy AND NOT fbOpen.bError THEN
        hFile := fbOpen.hFile;
        eState := 30;

    ELSIF fbOpen.bError THEN
        bError := TRUE;
        eState := 100;
    END_IF


// WRITE HEADER (FIRST-TIME ONLY)

30:
    IF NOT bHeaderWritten THEN
        
        sLine := 'Time,MirrorOffset,LaserOffset';
        sLine := CONCAT(sLine, sCRLF);

        fbWrite(
            hFile      := hFile,
            pWriteBuff := ADR(sLine),
            cbWriteLen := LEN(sLine),
            bExecute   := TRUE
        );

        bHeaderWritten := TRUE;
        eState := 31;

    ELSE
        ReadIndex := 0;
        eState := 40;
    END_IF


// WAIT HEADER WRITE

31:
    fbWrite(bExecute := FALSE);

    IF NOT fbWrite.bBusy AND NOT fbWrite.bError THEN
        ReadIndex := 0;
        eState := 40;
    END_IF


// WRITE LOG ENTRIES

40:
    fbWrite(bExecute := FALSE);

    IF ReadIndex < Count THEN
        
        index := (WriteIndex + 1000 - Count + ReadIndex) MOD 1000;

        // Build CSV row
        sLine := SYSTEMTIME_TO_STRING(aLog[index].tStamp);
        sLine := CONCAT(sLine, ',');
        sLine := CONCAT(sLine, LREAL_TO_STRING(aLog[index].Var1));
        sLine := CONCAT(sLine, ',');
        sLine := CONCAT(sLine, LREAL_TO_STRING(aLog[index].Var2));
        sLine := CONCAT(sLine, ',');
        sLine := CONCAT(sLine, INT_TO_STRING(aLog[index].Var3));
        sLine := CONCAT(sLine, sCRLF);

        fbWrite(
            hFile      := hFile,
            pWriteBuff := ADR(sLine),
            cbWriteLen := LEN(sLine),
            bExecute   := TRUE
        );

        eState := 41;

    ELSE
        eState := 50;
    END_IF


// WAIT LINE WRITE

41:
    fbWrite(bExecute := FALSE);

    IF NOT fbWrite.bBusy AND NOT fbWrite.bError THEN
        ReadIndex := ReadIndex + 1;
        eState := 40;   // Continue writing next entry
    END_IF


// CLOSE FILE

50:
    fbClose(hFile := hFile, bExecute := TRUE);
    eState := 60;


//WAIT CLOSE AND FINISH

60:
    fbClose(bExecute := FALSE);

    Count := 0;
    WriteIndex := 0;

    bBusy := FALSE;
    bDoneStatus := TRUE;

    eState := 0;


// ERROR

100:
    bBusy := FALSE;
    bError := TRUE;
    eState := 0;

END_CASE

END_FUNCTION_BLOCK

// ---- POUs/Sts/Datalog/FB_Datalogger3.TcPOU
FUNCTION_BLOCK FB_Datalogger3
VAR_INPUT
	iScaledTemp				: INT;
	sAssemblytype				: STRING;	//Needs to be set to the correct var in fb_stsAct, comes from st_recipe_assemblydata
	iStationIdDirect		: UDINT; // Station Id from strecipe assemblydata. 
	stMirrorData       		: REFERENCE TO ST_Vis_Mirror;
	stLaserData				: REFERENCE TO ST_Vis_Laser;
	fbHeaterControl			: REFERENCE TO FB_HeaterControl;
	stRecipeData			: reference TO ST_Recipe_AssemblyData;
                        	
    bEnable             	: BOOL;        // Rising edge = add one log entry
    bSave               	: BOOL;        // Rising edge = write CSV to a NEW timestamped file
	//istation				: INT :=8;
	stRecipeAssemblyData	: REFERENCE TO ST_Recipe_AssemblyData;
	fbStsAct				: REFERENCE TO FB_StsAct;
	
	//sMotTypeTest			: STRING := '7A6681';
//     Stepperpos          : LREAL;
//     SensorVal           : INT;
//     StepperHomed        : BOOL;
//     Var4                : BOOL;
//     Var5                : LREAL;
//     Var6                : INT;
//     Var7                : LREAL;
//     Var8                : BOOL;
//     Var9                : BOOL;
//     Error               : BOOL;
END_VAR

VAR_OUTPUT
    bBusy               	: BOOL;
    bDone               	: BOOL;
    bError              	: BOOL;
	bArrayWriteDone			: BOOL;
END_VAR                 	
                        	
VAR                     	
                        	
    aLog        			: ARRAY[0..999] OF ST_LogEntry;
    WriteIndex  			: UINT := 0;
    Count       			: UINT := 0;
    ReadIndex   			: UINT := 0;
                			
                			
    rEnable     			: R_TRIG;
    rSave       			: R_TRIG;
                			
                			
    fbOpen      			: FB_FileOpen;
    fbWrite     			: FB_FileWrite;
    fbClose     			: FB_FileClose;
                			
    hFile       			: UINT;
    sLine       			: STRING(255);
    sCRLF       			: STRING(2) := '$R$L'; // CRLF //Rivinvaihto
    // Base folder      	
    sBaseFolder 			: STRING(255) := 'C:\ProgramData\Beckhoff\TwinCAT\3.1\Boot\'; //Usbitikulle rassaus
    sFileName   			: STRING(255);		// Full path with timestamped filename
                        	
    index          			: UINT;
    eState         			: INT := 0;
                        	
                        	
    fbSysTime  				: FB_LocalSystemTime;
    CurrentDT  				: TIMESTRUCT;
                        	
                        	
    sSystemTime				: STRING(64);		//Full systemtime in string
	sTimeShort				: STRING (64);		//Shortened systemtime. Järjestelmäaika string josta millisekunnit pois
    pos        				: INT;
	iDot					: INT;				//Tunnistetaan piste sekuntien ja millis välissä
	            			
	MotorId					: STRING(64);		//Only for testing
	                    	
	WriteDoneTof			: TOF;
	DoneTof					: TOF;
	bDoneStatus				: BOOL;
	bWriteDone				: BOOL;
	
	//Station id variables
	sStationIdConvert 		: STRING;			//Asemanumeron kääntö stringiksi
	sStationID				: STRING;			//' _S'+Aseman numero stringinä
	sStationS				: STRING := '_S';	// S kirjain tiedostonimeen osoittamaan asemaa, turha? Voisi korvata '_S'
	sStationUnderScore		: STRING := '_';
	sFileNameStationId		: STRING;			// Final station id to be printed on the filename '_SX_'
	
	sFinalTimeString		: STRING;			// Aika stringinä, josta poistettu ms ja s
	SystemDT	:DT;
END_VAR

WriteDoneTof( IN := bWriteDone	, PT := T#0.2S, Q => bArrayWriteDone);
DoneTof(IN := bDoneStatus, PT := T#0.2S, Q => bDone);
bWriteDone := FALSE;
bDoneStatus := FALSE;


//Station id filename modification
sStationIDconvert := UDINT_TO_STRING (iStationIdDirect); //Käännetään asemanumero strngiksi
sStationID:=CONCAT(sStationS, sStationIDconvert); //Yhdistetään _S ja asemanumero string, syntyy _SX, jossa X asemanumero
sFileNameStationId := CONCAT (sStationID, sStationUnderScore); //Yhidstetään edellinen _SX ja alaviiva perään, syntyy _SX_


//  GET SYSTEM TIME from amsnetid
fbSysTime(sNetID :='192.168.1.11.1.1',		//192.168.1.11.1.1 //Asetettu testi-pcn amsnetid
					bEnable := TRUE);


// LOG 1 SET OF DATA WHEN bENABLE
rEnable(CLK := bEnable);

IF rEnable.Q AND NOT bBusy THEN

    aLog[WriteIndex].tStamp	:= fbSysTime.systemTime;
    aLog[WriteIndex].Var1	:= stMirrorData.rMirrorOffsetToCalPoints[1];  //stDetection.stMirror.rMirrorOffsetToCalPoints[1];
    aLog[WriteIndex].Var2	:= stLaserData.rLaserOffsetToSetPoint[0];     //stDetection.stLaser.rLaserOffsetToSetPoint[0];
    aLog[WriteIndex].Var3	:= iscaledtemp;                               //fbHeater.ScaledTemp;

    // Advance write pointer
    WriteIndex := WriteIndex + 1;
	bWriteDone := TRUE;
    IF WriteIndex > 999 THEN WriteIndex := 0; END_IF

    // Increment count to 1000
    IF Count < 1000 THEN Count := Count + 1; END_IF
END_IF



//bSave START NEW FILE WRITE 
rSave(CLK := bSave);

IF rSave.Q AND (Count > 0) AND (NOT bBusy) THEN
    
// Build filename
sSystemTime := SYSTEMTIME_TO_STRING(fbSysTime.systemTime);
//Remove millis from systemtime
iDot := FIND(sSystemTime, '.');
	IF iDot > 0 THEN
	    sTimeShort := LEFT(sSystemTime, iDot - 1);                  
	ELSE
	    sTimeShort := sSystemTime;                                   
	END_IF

// Convert : to -
FOR pos := 1 TO LEN(sTimeShort) DO
    IF sTimeShort[pos] = BYTE#58 THEN      // ':' ASCII 58
        sTimeShort[pos] := BYTE#45;        // replace with '-' ASCII 45
    END_IF
END_FOR;

// Convert  -  into _
sTimeShort[10] := BYTE#95;

sFinalTimeString := LEFT(sTimeShort, LEN(sTimeShort) - 3); //Removing seconds from the timestring

// Build final filename
sFileName := CONCAT(sBaseFolder, 'Log_');
sFileName := CONCAT(sfileName,sAssemblyType ); //Assemblynumero suoraan tähän stringinä, alaviiva logista ja asemanumerosta.
sFileName := CONCAT(sfileName,sFileNameStationId );  //Tähän viritetty station id _SX_.
sFileName := CONCAT(sFileName, sFinalTimeString); //aika ilman millis, hävitetään sekunnitkin?
sFileName := CONCAT(sFileName, '.csv');

    // Arm save sequence
    bBusy  := TRUE;
    bDone  := FALSE;
    bError := FALSE;
    eState := 10;
END_IF

//SAVE STATE MACHINE

CASE eState OF
    // Idle
    0: 
      
    // Open NEW filE
    10:
        fbOpen(
            sPathName := sFileName,
            nMode     := FOPEN_MODEWRITE,     // NEW FILE every save
            ePath     := PATH_GENERIC,
            bExecute  := TRUE
        );
        eState := 20;
    
    // Wait for file open
    20:
        fbOpen(bExecute := FALSE);

        IF NOT fbOpen.bBusy AND NOT fbOpen.bError THEN
            hFile := fbOpen.hFile;
            eState := 30;

        ELSIF fbOpen.bError THEN
            bError := TRUE;
            eState := 100;
        END_IF

    // Write header
    30:
        sLine := 'Time,MirrorOffset,LaserOffset';
        sLine := CONCAT(sLine, sCRLF);

        fbWrite(
            hFile      := hFile,
            pWriteBuff := ADR(sLine),
            cbWriteLen := LEN(sLine),
            bExecute   := TRUE
        );
        eState := 31;

    // Wait header write
    31:
        fbWrite(bExecute := FALSE);

        IF NOT fbWrite.bBusy AND NOT fbWrite.bError THEN
            ReadIndex := 0;
            eState := 40;
        END_IF

    //  Write data rows
    40:
        fbWrite(bExecute := FALSE);

        IF ReadIndex < Count THEN
            index := (WriteIndex + 1000 - Count + ReadIndex) MOD 1000; //MAKES SURE INDEX IS POSITIVE

            // Build CSV row
            sLine := SYSTEMTIME_TO_STRING(aLog[index].tStamp);  
            sLine := CONCAT(sLine, ',');
            sLine := CONCAT(sLine, LREAL_TO_STRING(aLog[index].Var1));
            sLine := CONCAT(sLine, ',');
            sLine := CONCAT(sLine, LREAL_TO_STRING(aLog[index].Var2));
            sLine := CONCAT(sLine, ',');
            sLine := CONCAT(sLine, INT_TO_STRING(aLog[index].Var3));
            sLine := CONCAT(sLine, sCRLF);

            fbWrite(
                hFile      := hFile,
                pWriteBuff := ADR(sLine),
                cbWriteLen := LEN(sLine),
                bExecute   := TRUE );

            eState := 41;

        ELSE
            eState := 50; // no more rows
        END_IF


    // Wait row write
    41:
        fbWrite(bExecute := FALSE);

        IF NOT fbWrite.bBusy AND NOT fbWrite.bError THEN
            ReadIndex := ReadIndex + 1;
            eState := 40;   // next row
        END_IF


    // Close file
    50:
        fbClose(hFile := hFile, bExecute := TRUE);
        eState := 60;

    // Finish & reset buffer
    60:
        fbClose(bExecute := FALSE);

        Count := 0;
        WriteIndex := 0;

        bBusy := FALSE;
        bDone := TRUE;
        eState := 0;
   
    100:
        bBusy := FALSE;
        bError := TRUE;
        eState := 0;

END_CASE

END_FUNCTION_BLOCK

// ---- POUs/Sts/FB_HeaterControl.TcPOU
FUNCTION_BLOCK FB_HeaterControl
VAR_INPUT
	bExecuteTest		: BOOL;
	stPlcCom			: REFERENCE TO	ST_Sts_PlcCom;
	stModulePlcCom		: REFERENCE TO ST_Module_PlcCom;
	bHeatingOnOff		: BOOL;
	bResetHeating		: BOOL;
	iStationId			: UDINT;
END_VAR
VAR_OUTPUT
	bTempReached		: BOOL := TRUE;
	bTestTempReached	: BOOL;
	ScaledTemp			: INT;
	bHeatingFailed		: BOOL;
END_VAR
VAR
	HeaterState			: INT :=0;
	HeatingTmr : TON;
	StartTmr : TON;
	iHeatingTime		: INT;
	iOffTime			: INT;
END_VAR


////////////////////////////////////////////////////////////
///////////////////////////////////////////////////////////////////
IF NOT stModulePlcCom.stPlcComIn.bEstopOk THEN
	HeaterState := 999;
	END_IF
		

ScaledTemp := (stPlcCom.stPlcComIn.PtcRawTemp / 10);

StartTmr( PT := UDINT_TO_TIME(iStationId * 2000));

IF NOT bHeatingOnOff AND NOT bExecuteTest AND stModulePlcCom.stPlcComIn.bEstopOk THEN
	HeaterState :=0;
	StartTmr.in:= FALSE;
END_IF

IF HeaterState >= 10 AND stPlcCom.stPlcComIn.PtcRawTemp >= 550 THEN
	bHeatingFailed := TRUE;
	HeaterState :=1000;
END_IF
// estoppi, jos heatingonoff false niin kaikki 0



CASE HeaterState OF
	0:	IF stModulePlcCom.stPlcComIn.bEstopOk THEN
			stPlcCom.stPlcComOut.bHeaterFan := FALSE;
			stPlcCom.stPlcComOut.bHeaterElement := FALSE;
			IF bHeatingOnOff THEN		// AND StartTmr.Q
				StartTmr.IN := TRUE;
				HeaterState := 5; //Ajastin päälle kun lämmitin tulille
			ELSIF bExecuteTest THEN
				 HeaterState := 5000;
			END_IF
		ELSE
			StartTmr.IN := FALSE;
			stPlcCom.stPlcComOut.bHeaterFan := FALSE;
			stPlcCom.stPlcComOut.bHeaterElement := FALSE;
			HeaterState := 0;	
		END_IF
		
	5:
		IF bHeatingOnOff AND StartTmr.Q THEN
			stPlcCom.stPlcComOut.bHeaterFan := TRUE;  //Ajastin päälle kun lämmitys päälle, ajastimen jälkeen lömmitin oikeasti tulille. Ajstimen nollaus kun lämmituys loppuu.
			StartTmr.IN := FALSE;
			HeaterState := 10;
		END_IF
	
	10:
		IF StPlcCom.stPlcComIn.PtcRawTemp <= 470 THEN
			iHeatingTime := 16;
			iOffTime := 4;
		ELSIF StPlcCom.stPlcComIn.PtcRawTemp <= 490 THEN
			iHeatingTime := 12;
			iOffTime := 8;
		ELSIF StPlcCom.stPlcComIn.PtcRawTemp <= 510 THEN
			iHeatingTime := 8;
			iOffTime := 12;
		ELSIF StPlcCom.stPlcComIn.PtcRawTemp <= 530 THEN
			iHeatingTime := 4;
			iOffTime := 16;
		END_IF
		HeaterState := 20;
			
	20:

		IF HeatingTmr.Q THEN
			HeatingTmr(IN:=FALSE);
			stPlcCom.stPlcComOut.bHeaterElement := FALSE;
			HeaterState := 30;
		ELSE
			HeatingTmr(IN:=TRUE,PT:=INT_TO_TIME(iHeatingTime*1000));
		END_IF
		
	30:
		IF HeatingTmr.Q THEN
			HeatingTmr(IN:=FALSE);
			stPlcCom.stPlcComOut.bHeaterElement := TRUE;
			HeaterState := 10;
		ELSE
			HeatingTmr(IN:=TRUE, PT:= INT_TO_TIME(iOffTime*1000));
		END_IF
		
	999:
		bHeatingOnOff := FALSE;
		stPlcCom.stPlcComOut.bHeaterElement := FALSE;
		stPlcCom.stPlcComOut.bHeaterFan:= FALSE;
		HeatingTmr(IN:=FALSE);
		StartTmr.IN := FALSE;
		bExecuteTest := FALSE;
			
	1000:
		bHeatingOnOff := FALSE;
		stPlcCom.stPlcComOut.bHeaterElement := FALSE;
		stPlcCom.stPlcComOut.bHeaterFan:= FALSE;
		
		IF bResetHeating THEN
			bHeatingFailed :=FALSE;
			HeaterState := 0;
		END_IF
		
//HeaterTestFunction				
	5000:
		stPlcCom.stPlcComOut.bHeaterFan := TRUE;
		IF bExecuteTest THEN
			HeaterState := 5010;
		ELSE
			HeaterState := 5000;	
		END_IF
	
	5010:
		IF stPlcCom.stPlcComIn.PtcRawTemp <= 280 THEN
				stPlcCom.stPlcComOut.bHeaterElement := TRUE;
				bTestTempReached :=FALSE;
				
			ELSIF StPlcCom.stPlcComIn.PtcRawTemp >= 280 THEN
				stPlcCom.stPlcComOut.bHeaterElement := FALSE;
				stPlcCom.stPlcComOut.bHeaterFan := FALSE;
				bTestTempReached := TRUE;
				bExecuteTest := FALSE;
				HeaterState := 5000;	
		END_IF
	
END_CASE

END_FUNCTION_BLOCK

// ---- POUs/Sts/FB_StsAct.TcPOU
FUNCTION_BLOCK FB_StsAct
VAR_IN_OUT
	bActivateStation : BOOL;
END_VAR
VAR_INPUT
	stLaserData	: REFERENCE TO ST_Vis_Laser;
	stMirrorData : REFERENCE TO ST_Vis_Mirror;
	stModuleHmi	: REFERENCE TO ST_ModuleHmi;
	stModulePlcCom	: REFERENCE TO ST_Module_PlcCom;

	bEngageSlider	:  BOOL;
	bEngageHolder : BOOL;
	bRobotReadyForStation : BOOL;
	bDismountingDone : BOOL;
	bAdjDone: BOOL;
	iStationId	: UDINT;
	rAssemblyCuringTime : REAL := 1; // IN HOURS
	bAllowStart : BOOL;
	iAdjustmentCount : INT;
	bReleaseHolders : BOOL;
END_VAR
VAR_OUTPUT
	bTrigPosCam		: BOOL;
	bTrigAngCam		: BOOL;
	bTrigPosCamLightTest	: BOOL; // triggaa testiohjelman kameralle joka katsoo että laseri, taustavalo ja itse kamera toimii. Palaute tieto on stDetectionData.stMirror.bImagingStatusOk
	bTrigPosCamLaserTest : BOOL;
	bTrigPosCamCoupler : BOOL;
	bInHoldForRobot : BOOL;
	rRobotAdjValue	: LREAL;
	bStationChecksPassed : BOOL;
	bCheckDone : BOOL;
	bHoldRobotForAdj : BOOL;
	bAssemblyFailed	: BOOL;


	sTimeLeft		: STRING;
	bDisabledByCycleDone	: BOOL;
	bPlacingDone	: BOOL;
END_VAR
VAR
	stPlcCom	: ST_Sts_PlcCom;
	fbStepper	: FB_Stepper;
	fbHeater 	: FB_HeaterControl;
	fbHeater2:	FB_CuringStationHeaterControl;
	eStationState	: E_StsActState;
	stRecipe		:ST_Recipe_AssemblyData;
	fbEventLogger		: FB_EventLogger;
	
	// PROPERTIES
	bMotorInStation	: BOOL;
	bAllPartsInStation : BOOL;
	bStationDone : BOOL;
	// MOTOR MOTION COMMANDS
	bStepForward: BOOL;
	bStepBackwards : BOOL;
	bExecuteAdj : BOOL;
	
	//INTERNAL STATUS VARIABLES
	bDetectionRetry: BOOL;
	rDetectedOffset	: LREAL;
	bLastDatalog	: BOOL;
	iStatus2Cycles	: UINT;
	bInitialStartup	: BOOL;
	bResetStation	: BOOL;
	bSetOnce : BOOL;
	bEstopCycled	: BOOL;
	iErrorId		: INT;
	sErrorId		: STRING;
	tTimeLeft		: TIME;
	iDot			: INT;
	sTime			: STRING;
	
	// CASE STEP HANDLERS
	iAssemblyCheckStep	: INT;
	iPosAdjStep			: INT;
	iStartupCheckStep	: INT;
	iStatus2Step		: INT;
	iDatalogStep		: INT;
	iMountingStep		: INT;
	
	// STATUS VARIABLES
	iAssemblyStatus : INT; // IF CURING HAS JUST BEGUN STATUS IS 1. WHEN FIRST ACCEPTED CHECK HAS OCCURED STATUS IS 2. WHEN ASSEMBLY HAS REACHED 30 MIN ACCEPETED TIME STATUS IS 3. WHEN STS IS EMPTY STATUS IS 0.
	// TIMERS
	StartupCheckTmr : TON;
	StartupStartTmr : TON;
	DataloggingTmr1 : TON;
	DataloggingTmr2	: TON;
	AssemblyDoneTmr : TON;
	bImagingTmr : TON;
	AxisResetTmr	: TON;
	MountingTmr	: TON;
	MoveTmr	: TON;
	
	fbdatalogger2		: FB_Datalogger2;
	fbdatalogger3		: FB_Datalogger3;
	
END_VAR

fbHeater(stPlcCom := stPlcCom, iStationId := iStationId, stModulePlcCom := stModulePlcCom);
fbStepper(rStepperVel := 10, stPlcCom := stPlcCom, bEstopOk := stModulePlcCom.stPlcComIn.bEstopOk);
StartupCheckTmr(PT := T#120S);
StartupStartTmr(PT := UDINT_TO_TIME(iStationId * 4 * 1000));
AssemblyDoneTmr(PT := REAL_TO_TIME(rAssemblyCuringTime * 60 * 60 * 1000));
DataloggingTmr1(PT := T#2M);
DataloggingTmr2(PT := T#5M);
bImagingTmr(PT := T#1.5S);
AxisResetTmr(PT:= T#5S);
fbdatalogger2(stMirrorData := stMirrorData, stLaserData := stLaserData, iScaledTemp := fbHeater.ScaledTemp);
fbdatalogger3(stMirrorData:=stMirrorData, stLaserData :=stLaserData, iScaledTemp := fbHeater.ScaledTemp, stRecipeAssemblyData:=stRecipe,iStationIdDirect:=iStationId, sAssemblytype:=stRecipe.sAssemblyType );
MountingTmr(PT := T#5S);
MoveTmr(PT := T#5S);
fbEventLogger(sErrorCode := sErrorId, stModuleHmi := stModuleHmi);
tTimeLeft := AssemblyDoneTmr.PT - AssemblyDoneTmr.ET;
sTime := (TIME_TO_STRING(tTimeLeft));


iDot := FIND(sTime, '.');
IF iDot > 0 THEN
	sTimeLeft := LEFT(sTime, iDot - 1);                                                  
END_IF

IF NOT stModulePlcCom.stPlcComIn.bEstopOk THEN
	eStationState := E_StsActState.Disabled;
	bEstopCycled := TRUE;
ELSIF bEstopCycled THEN
	bEstopCycled := FALSE;
	bResetStation := TRUE;
ELSIF NOT bActivateStation THEN
	eStationState := E_StsActState.Disabled;
END_IF

IF stModuleHmi.bModuleProductionStop THEN
	eStationState := E_StsActState.HoldForValveRelease;
END_IF

CASE eStationState OF
	E_StsActState.StartupCheck:	
		CASE iStartupCheckStep OF
			0: bStationChecksPassed := FALSE;
				bActivateStation := TRUE;
				bDisabledByCycleDone := FALSE;
				bSetOnce := TRUE;
				bCheckDone := FALSE;
					IF stModulePlcCom.stPlcComIn.bEstopOk AND stModulePlcCom.stPlcComIn.bSafetyOk THEN
						IF NOT bInitialStartup THEN
							IF stModuleHmi.bModuleStartup THEN
								StartupStartTmr.IN := TRUE;
								bInitialStartup := TRUE;
							END_IF
						ELSE
							StartupStartTmr.IN := TRUE;
						END_IF
					END_IF
				IF StartupStartTmr.Q THEN
					iStartupCheckStep := 1;
				END_IF
			1:	IF fbStepper.bAxisReady THEN
					AxisResetTmr.IN := FALSE;
					fbStepper.bResetAxis := FALSE;
					iStartupCheckStep := 2;
				ELSIF fbStepper.bError THEN
					fbStepper.bResetAxis := TRUE;
					AxisResetTmr.IN := TRUE;
				ELSIF AxisResetTmr.Q THEN
					eStationState := E_StsActState.Disabled;
					AxisResetTmr.IN := FALSE;
				END_IF
				
			2:	StartupCheckTmr.IN := TRUE;
				fbStepper.bExecuteEncHoming := TRUE;
				fbHeater.bExecuteTest := TRUE;
				iStartupCheckStep := 3;
			3: 
				IF stPlcCom.stPlcComIn.bGripperHomeSensor AND NOT stPlcCom.stPlcComIn.bSliderHomeSensor THEN
					bTrigPosCamLightTest := TRUE;
					bTrigPosCam := TRUE;
					stPlcCom.stPlcComOut.bUnderLight := TRUE;
					iStartupCheckStep := 4;
				ELSE
					stPlcCom.stPlcComOut.bGripper := TRUE;
					stPlcCom.stPlcComOut.bPusher := TRUE;
				END_IF
			4: IF stMirrorData.bLightTestOk THEN
					bTrigPosCamLightTest := FALSE;
					bTrigPosCam := FALSE;
					IF NOT stMirrorData.bImagingDone THEN
						iStartupCheckStep := 5;
					END_IF
				ELSIF stMirrorData.bDetectionFailed THEN
					bTrigPosCamLightTest := FALSE;
					bTrigPosCam := FALSE;
					eStationState := E_StsActState.Disabled;
					iErrorId := 305;
					sErrorId := CONCAT(CONCAT('3', UDINT_TO_STRING(iStationId)), '5');
					fbEventLogger.bRaiseAlarm[12]:= TRUE;
				END_IF
			5: stPlcCom.stPlcComOut.bUnderLight := FALSE;
				bTrigPosCamLaserTest := TRUE;
				IF stMirrorData.bReadyForTrigger THEN
					bTrigPosCam := TRUE;
					iStartupCheckStep := 6;
				END_IF
				
			6: IF stMirrorData.bLaserTestOk THEN
					bTrigPosCamLaserTest := FALSE;
					bTrigPosCam := FALSE;
					IF NOT stMirrorData.bImagingDone THEN
						iStartupCheckStep := 7;
					END_IF
				ELSIF stMirrorData.bDetectionFailed THEN
					bTrigPosCam := FALSE;
					eStationState := E_StsActState.Disabled;
					bTrigPosCamLaserTest := FALSE;
					fbEventLogger.bRaiseAlarm[13] := TRUE;
					sErrorId := CONCAT(CONCAT('3', UDINT_TO_STRING(iStationId)), '6');
					iErrorId := 306;
				END_IF 
 			7: IF fbStepper.bAxisReady AND fbStepper.bEnchomingDone THEN
					iStartupCheckStep := 8;
				ELSIF fbStepper.bError THEN
					eStationState := E_StsActState.Disabled;
					iErrorId := 300; // lisää muuttujan fbStepper.nErrorID tekstiin
					sErrorId := CONCAT(CONCAT(CONCAT('3', UDINT_TO_STRING(iStationId)), '5'), UDINT_TO_STRING(fbStepper.nErrorID));			//OLi CONCAT(CONCAT('3', INT_TO_STRING(iStationId)), '0');
					fbEventLogger.bRaiseAlarm[8]:= TRUE;	//StepperError?
				END_IF
				
			8: IF fbHeater.bTestTempReached THEN
					fbHeater.bExecuteTest := FALSE;
					iStartupCheckStep := 9; 
				END_IF
				
			9: bStationChecksPassed := TRUE;
				bCheckDone := TRUE;
				eStationState := E_StsActState.Idle; // VAIHDA IDLEEN
				iStartupCheckStep := 0;
			
		END_CASE
		IF StartupCheckTmr.Q THEN
			IF iStartupCheckStep > 6 THEN
				eStationState := E_StsActState.Disabled;
				iErrorId := 302;
				sErrorId := CONCAT(CONCAT('3', UDINT_TO_STRING(iStationId)), '2');
				fbEventLogger.bRaiseAlarm[10]:= TRUE;
			ELSIF iStartupCheckStep <= 3 THEN
				eStationState := E_StsActState.Disabled;
				iErrorId := 301;
				sErrorId := CONCAT(CONCAT('3', UDINT_TO_STRING(iStationId)), '1');
				fbEventLogger.bRaiseAlarm[9]:= TRUE;
			END_IF
		END_IF
		
	E_StsActState.AssemblyCheck:
		CASE iAssemblyCheckStep OF
			0: CASE iAssemblyStatus OF
				0: eStationState := E_StsActState.Idle;
				1: iAssemblyCheckStep := 1;
				2: bPlacingDone := TRUE;
					 CASE iStatus2Step OF
						0: DataloggingTmr1.IN := TRUE;
							iStatus2Step := 1; 
						1: 	IF DataloggingTmr1.Q  AND iStatus2Cycles < 15 THEN
								DataloggingTmr1.IN := FALSE;
								iStatus2Step := 2;
							ELSIF iStatus2Cycles >= 15 THEN
								iAssemblyStatus := 3;
								iStatus2Cycles := 0;
								DataloggingTmr1.IN := FALSE;
							END_IF
							
						2: iStatus2Cycles := iStatus2Cycles +1;
							iStatus2Step := 0;
							iAssemblyCheckStep := 1;
					END_CASE
				3: IF AssemblyDoneTmr.Q THEN
						iAssemblyStatus := 4;
						iAssemblyCheckStep := 1;
						bLastDatalog := TRUE;
					ELSE
						DataloggingTmr2.IN := TRUE;
						IF DataloggingTmr2.Q THEN
							iAssemblyCheckStep := 1;
							DataloggingTmr2.IN := FALSE;
						END_IF
					END_IF
				4: eStationState := E_StsActState.RobotSlotHold;
					bStationDone := TRUE;
			END_CASE
			
			
			1: stPlcCom.stPlcComOut.bUnderLight := TRUE;
				bTrigPosCam := TRUE;
				iAssemblyCheckStep := 2;
			2:	IF stMirrorData.bImagingDone THEN	
					bTrigPosCam := FALSE;
					iAssemblyCheckStep := 3;
					stPlcCom.stPlcComOut.bUnderLight := FALSE;
				ELSIF stMirrorData.bDetectionFailed THEN
					IF NOT bDetectionRetry THEN
						bTrigPosCam := FALSE;
						iAssemblyCheckStep := 1;
						bDetectionRetry := TRUE;
					ELSE
						iErrorId := 1106; // ERROR CODES NOT CREATED, This error tells that detection failed twice in current station.
						Err.Err;
						eStationState := E_StsActState.Disabled;
					END_IF
				END_IF
				
			3:	IF iAssemblyStatus = 1 THEN
					IF iAdjustmentCount < 10 THEN
						IF stMirrorData.rMirrorOffsetToCalPoints[1] > 0.01 OR stMirrorData.rMirrorOffsetToCalPoints[1] < -0.01 THEN
							eStationState := E_StsActState.RobotSlotHold;
							iAssemblyCheckStep := 0;
							bDetectionRetry := FALSE;
						ELSE
							bHoldRobotForAdj := FALSE;
							iAssemblyCheckStep := 4;
						END_IF
					ELSE
						bAssemblyFailed := TRUE;
					END_IF
				ELSE 
					iAssemblyCheckStep := 4;
				END_IF
				
			4: bImagingTmr.IN := TRUE;
				IF bImagingTmr.Q THEN
					bTrigAngCam := TRUE;
					bImagingTmr.IN := FALSE;
					iAssemblyCheckStep := 5;
				END_IF
			5: IF stLaserData.bImagingDone THEN
					bTrigAngCam := FALSE;
					iAssemblyCheckStep := 6;
				ELSIF stLaserData.bDetectionFailed THEN
					IF NOT bDetectionRetry THEN
						bTrigAngCam := FALSE;
						iAssemblyCheckStep := 4;
						bDetectionRetry := TRUE;
					ELSE
						iErrorId := 1106; // ERROR CODES NOT CREATED, This error tells that detection failed twice in current station.
						Err.Err;
						eStationState := E_StsActState.Disabled;
					END_IF
				END_IF
			6:	IF iAssemblyStatus <= 2 THEN
				
					MoveTmr.IN := TRUE;
					IF stLaserData.rLaserOffsetToSetPoint[0] < -5 THEN 
						rDetectedoffset := (stLaserData.rLaserOffsetToSetPoint[0]/10);
						bStepForward := TRUE;
						IF MoveTmr.Q THEN
							eStationState := E_StsActState.AngleAdj;
							MoveTmr.IN := FALSE;
							iAssemblyCheckStep := 4;
							bDetectionRetry := FALSE;
						END_IF
					ELSIF stLaserData.rLaserOffsetToSetPoint[0] > 5 THEN
						rDetectedoffset := (stLaserData.rLaserOffsetToSetPoint[0]/10);
						bStepBackwards := TRUE;
						eStationState := E_StsActState.AngleAdj;
						iAssemblyCheckStep := 4;
						bDetectionRetry := FALSE;
					ELSE
						iAssemblyCheckStep := 7;
					END_IF
				ELSE
					iAssemblyCheckStep := 8;
				END_IF
				stLaserData.bImagingDone := FALSE;
				
			7:	iAssemblyStatus := 2;
				iAssemblyCheckStep := 8;
			8: eStationState := E_StsActState.DataLogging;
				iAssemblyCheckStep := 0;

		END_CASE
	
	E_StsActState.Idle:
		IF stModuleHmi.bModuleProductionStart AND bAllowStart AND bStationChecksPassed THEN
			eStationState := E_StsActState.RobotSlotHold;
		END_IF
		
		
	E_StsActState.AngleAdj:
		IF fbStepper.bAxisReady THEN
			IF bStepForward THEN
				fbStepper.rStepCount := rDetectedoffset;
				IF fbStepper.rStepCount = rDetectedoffset THEN
					fbStepper.bStepForward := TRUE;
					bStepForward := FALSE;
				END_IF
			ELSIF bStepBackwards THEN
				fbStepper.rStepCount := rDetectedoffset;
				fbStepper.bStepBackward := TRUE;
				bStepBackwards := FALSE;
			END_IF
			IF fbStepper.bDone THEN
				eStationState := E_StsActState.AssemblyCheck;
			END_IF
		END_IF
		
	E_StsActState.RobotSlotHold:
		IF bRobotReadyForStation THEN
			bInHoldForRobot := FALSE;
			IF NOT bMotorInStation THEN
				eStationState := E_StsActState.ProductMounting;
			ELSIF bAllPartsInStation AND NOT bStationDone THEN
				eStationState := E_StsActState.PositionAdj;
			ELSIF bStationDone THEN
				eStationState := E_StsActState.ProductDisMounting;
			END_IF
		ELSE
			bInHoldForRobot := TRUE;
		END_IF
		
	E_StsActState.PositionAdj:
		CASE iPosAdjStep OF
		0: rRobotAdjValue := stMirrorData.rMirrorOffsetToCalPoints[1];
			iPosAdjStep := 1;
		1: bExecuteAdj := TRUE;
			iPosAdjStep := 2;
		2: IF bAdjDone THEN
				bExecuteAdj := FALSE;
				iPosAdjStep := 0;
				iAdjustmentCount := iAdjustmentCount +1;
				eStationState := E_StsActState.AssemblyCheck;
				bAdjDone := FALSE;
			END_IF
		END_CASE
		
	E_StsActState.ProductMounting: // LISÄÄ ANTURITARKISTUKSET
		CASE iMountingStep OF
			0: IF bEngageHolder THEN
					stPlcCom.stPlcComOut.bGripper := FALSE;
					bMotorInStation := TRUE;
					iMountingStep := 1;
				ELSE
					stPlcCom.stPlcComOut.bGripper := TRUE;
				END_IF
			1: stPlcCom.stPlcComOut.bUnderLight := TRUE;
				stPlcCom.stPlcComOut.bPusher := FALSE;
				bImagingTmr.IN := TRUE;
				iMountingStep := 2;
			2: IF bImagingTmr.Q THEN
					bTrigPosCamCoupler := TRUE;
					bImagingTmr.IN := FALSE;
					bTrigPosCam := TRUE;
					iMountingStep := 3;
				END_IF
			3: 	IF stMirrorData.bImagingDone THEN
					bTrigPosCamCoupler := FALSE;
					stPlcCom.stPlcComOut.bPusher := TRUE;
					bTrigPosCam := FALSE;
					iMountingStep := 4;
				END_IF
			4:IF bEngageSlider AND NOT stPlcCom.stPlcComIn.bSliderHomeSensor THEN
					stPlcCom.stPlcComOut.bPusher := FALSE;
					bAllPartsInStation := TRUE;
					bHoldRobotForAdj := TRUE;
					iMountingStep := 5;
				END_IF
				 
			5: 	IF bEngageHolder AND bEngageSlider THEN
					fbHeater.bHeatingOnOff := TRUE;
					AssemblyDoneTmr.IN := TRUE;
					MountingTmr.IN := TRUE;
					IF MountingTmr.Q THEN
						iMountingStep := 0;
						eStationState := E_StsActState.AssemblyCheck;
						MountingTmr.IN := FALSE;
						iAssemblyStatus := 1;
					END_IF
				END_IF
		END_CASE
		
		
	
	E_StsActState.ProductDisMounting:
		IF NOT bEngageHolder THEN
			stPlcCom.stPlcComOut.bGripper := TRUE;
		END_IF
		IF NOT bEngageSlider THEN
			stPlcCom.stPlcComOut.bPusher := TRUE;
		END_IF
		IF bDismountingDone THEN
			bDisabledByCycleDone := TRUE;
			eStationState := E_StsActState.Disabled;
			bMotorInStation := FALSE;
			bAllPartsInStation := FALSE;
			bDismountingDone := FALSE;
		END_IF
		
		
		
	E_StsActState.DataLogging:
		CASE iDatalogStep OF
			0: fbdatalogger3.bEnable := TRUE;
				iDatalogStep := 1;
			1: 	IF fbdatalogger3.bArrayWriteDone THEN
					fbdatalogger3.bEnable := FALSE;
					iDatalogStep := 2;
				END_IF
			
			2: 	IF bLastDataLog THEN
				// fbDatalogger.bSave := TRUE;
				 fbdatalogger3.bSave := TRUE;
				// fbdatalogger3.bSave :=TRUE;
				IF fbdatalogger3.bDone THEN
					 fbdatalogger3.bSave :=FALSE;
					 bLastDataLog := FALSE;
				 END_IF
				 // OKSENNA DATA TIEDOSTOON
			ELSE
				fbdatalogger3.bEnable := FALSE;
				iDatalogStep := 0;
				eStationState := E_StsActState.AssemblyCheck;
			END_IF
		END_CASE
		
	E_StsActState.HoldForValveRelease:
		IF bReleaseHolders THEN
			stPlcCom.stPlcComOut.bGripper := TRUE;
			stPlcCom.stPlcComOut.bPusher := TRUE;
			bDisabledByCycleDone := TRUE;
			bReleaseHolders := FALSE;
			eStationState := E_StsActState.Disabled;
		END_IF
	
	E_StsActState.Disabled:
		Initialize();
		fbStepper.Initialize();
		bCheckDone := TRUE;
		IF bSetOnce THEN
			bActivateStation := FALSE;
			bSetOnce := FALSE;
		END_IF
		IF bResetStation OR bActivateStation THEN
			fbStepper.bResetAxis := TRUE;
			eStationState := E_StsActState.StartupCheck;
			bResetStation := FALSE;
		END_IF
		
END_CASE

PROPERTY AllPartsInStation : BOOL
GET
AllPartsInStation := bAllPartsInStation;
END_GET
SET
bAllPartsInStation := AllPartsInStation;
END_SET
END_PROPERTY

PROPERTY AssemblyDone : BOOL
GET
AssemblyDone := bStationDone;
END_GET
SET
bStationDone := AssemblyDone;
END_SET
END_PROPERTY

PROPERTY bHolderSensor : BOOL
GET
bHolderSensor := stPlcCom.stPlcComIn.bGripperHomeSensor;
END_GET
END_PROPERTY

PROPERTY bSliderSensor : BOOL
GET
bSliderSensor := stPlcCom.stPlcComIn.bSliderHomeSensor;
END_GET
END_PROPERTY

METHOD Initialize : BOOL
VAR_INPUT
END_VAR
	StartupStartTmr.IN := FALSE;
	iAssemblyStatus := 0;
	iDatalogStep := 0;
	iAssemblyCheckStep := 0;
	fbHeater.bHeatingOnOff := FALSE;
	fbHeater.bExecuteTest := FALSE;
	fbdatalogger3.bEnable := FALSE;
	fbdatalogger3.bSave := FALSE;
	StartupStartTmr.IN := FALSE;
	AssemblyDoneTmr.IN := FALSE;
	DataloggingTmr1.IN := FALSE;
	DataloggingTmr2.IN := FALSE;
	bImagingTmr.IN := FALSE;
	stPlcCom.stPlcComOut.bUnderLight := FALSE;
	bTrigPosCam := FALSE;
	bTrigAngCam := FALSE;
	bStationChecksPassed := FALSE;
	bStationDone := FALSE;
	bAllPartsInStation := FALSE;
	bMotorInStation := FALSE;
	bStepForward := FALSE;
	bStepBackwards := FALSE;
	bLastDatalog := FALSE;
	iStatus2Cycles := 0;
	bDetectionRetry := FALSE;
	iPosAdjStep	:= 0;
	iStartupCheckStep := 0;
	iStatus2Step := 0;
	bTrigPosCamLightTest := FALSE;
	bTrigPosCamLaserTest := FALSE;
	StartupCheckTmr.IN := FALSE;
	stMirrorData.bLightTestOk := FALSE;
	stMirrorData.bLaserTestOk := FALSE;
	iMountingStep := 0;
	iAdjustmentCount := 0;
	bHoldRobotForAdj := FALSE;
	bPlacingDone := FALSE;
END_METHOD

PROPERTY MotorInStation : BOOL
GET
MotorInStation := bMotorInStation;
END_GET
SET
bMotorInStation := MotorInStation;
END_SET
END_PROPERTY

END_FUNCTION_BLOCK

// ---- POUs/Sts/FB_Stepper.TcPOU
FUNCTION_BLOCK FB_Stepper
VAR_INPUT
	bStepForward				: BOOL;
	bStepBackward				: BOOL;
	rStepperVel					: LREAL;
	rStepCount					: LREAL := 1;
	bExecuteEncHoming			: BOOL;
	bResetAxis					: BOOL;
	stPlcCom					: REFERENCE TO ST_Sts_PlcCom;
	bInitializeAngle			: BOOL;
	bAutoReset					: BOOL;
	bEstopOk					: REFERENCE TO BOOL;
END_VAR
VAR_OUTPUT
	bAxisReady					: BOOL;
	rPosition					: LREAL;
	bAxisInitialized			: BOOL;
	bEnchomingDone				: BOOL;
	bDone						: BOOL;
	bError						: BOOL;
	nErrorID					: UDINT;
END_VAR
VAR
	fbAxis						: Axis_REf;
	fbJog						: MC_Jog;
	fbJogCont					: MC_Jog;
	fbHalt						: MC_Halt;
	fbStop						: MC_Stop;
	fbHome						: MC_Home;
	bAxis1StatusOk				: BOOL;
	
	rStepCountAct				: LREAL;
	
	bOperational				: BOOL;
	bExecuteHoming				: BOOL;
	iEncHomingStep				: INT;
	bJogForwardCont				: BOOL;
	bJogForward					: BOOL;
	bMovementStarted			: BOOL;
	bJogBackwards				: BOOL;
	bJogBackwardsCont			: BOOL;
	eState						: E_StepperState;
	fbReset						: MC_Reset;
	fbPower						: MC_Power;
	fbMoveAbs					: MC_MoveAbsolute;
	fbReadPos					: MC_ReadActualPosition;
	StopTmr						: TON;
	DoneTmr						: TOF;
	iInitializingStep 			: INT;
	bExecuteMoveAbs				: BOOL;
	rStepperDec						: LREAL := 14000;
	rStepperAcc						: LREAL := 14000;
END_VAR

fbAxis.ReadStatus();
StopTmr(PT := T#1S);
fbReadPos(Axis := fbAxis,Enable := TRUE, Position => rPosition);
DoneTmr(PT := T#0.5S, Q => bDone);
IF NOT bEstopOk THEN
	eState := E_StepperState.Error;
END_IF
DoneTmr.IN := FALSE;

CASE eState OF
	E_StepperState.Offline:
		bOperational := FALSE;
		IF NOT fbReset.Busy THEN
			IF NOT fbPower.Error AND NOT fbJog.Error AND NOT fbReset.Error AND NOT fbHalt.Error THEN
				bError := FALSE;
				bResetAxis := FALSE;
				IF NOT fbPower.Active OR NOT fbPower.enable THEN
					eState := E_StepperState.Power;
				ELSE
					eState := E_StepperState.Operational;
				END_IF
			ELSE
				eState := E_StepperState.Reset;
			END_IF
		END_IF
		 
	E_StepperState.Reset:
		bJogForward := FALSE;
		bJogForwardCont := FALSE;
		bJogBackwards := FALSE;
		bJogBackwardsCont := FALSE;
		fbReset.Execute := TRUE;		
		IF NOT fbReset.Busy AND fbReset.Done THEN
			fbPower.Enable:= FALSE;	
			fbReset.Execute := FALSE;
			eState := E_StepperState.Offline;
		ELSE
			eState := E_StepperState.Error;
		END_IF
	
	
	E_StepperState.Power:
		IF NOT bAxis1StatusOk THEN
			fbPower.Enable:= TRUE;
		END_IF
		IF bAxis1StatusOk THEN
			eState := E_StepperState.Operational;
		END_IF
		IF fbPower.Error THEN
			eState := E_StepperState.Offline;	
		END_IF
		
	E_StepperState.Operational:
		bOperational := TRUE;
		bAxisReady := TRUE;
		IF NOT bAxis1StatusOk OR bResetAxis THEN
			eState := E_StepperState.Offline;
		ELSIF bStepForward OR bStepBackward THEN
			eState := E_StepperState.Jog;
		ELSIF bExecuteEncHoming THEN
			eState := E_StepperState.EncHoming;
		ELSIF bInitializeAngle THEN
			eState := E_StepperState.Homing;
		END_IF
		
		
	E_StepperState.EncHoming:
		bAxisReady := FALSE;
			CASE iEncHomingStep	OF
				0: IF stPlcCom.stPlcComIn.bAngleMotorSensor THEN
						bJogForwardCont := FALSE;
						StopTmr.IN := TRUE;
						iEncHomingStep := 1;
					ELSE
						bJogForwardCont := TRUE;
					END_IF
					IF fbJog.Error OR bError THEN
						eState := E_StepperState.Error;
					END_IF
				1: IF StopTmr.Q THEN
					IF NOT bEnchomingDone THEN
						bExecuteHoming := TRUE;
						bExecuteEncHoming := FALSE;
					END_IF
					IF fbHome.Done THEN
						StopTmr.IN := FALSE;
						bExecuteHoming := FALSE;
						bEnchomingDone := TRUE;
						iEncHomingStep := 2;
					ELSIF fbHome.Error OR bError THEN
						eState := E_StepperState.Error;
					END_IF
				END_IF
				2: bJogForward := FALSE;
					eState := E_StepperState.Operational;
					bAxisInitialized := TRUE;
					iEncHomingStep := 0;
			END_CASE
			
			
	E_StepperState.Homing:
			bAxisReady := FALSE;
			CASE iInitializingStep OF
				0: IF bInitializeAngle THEN
						IF stPlcCom.stPlcComIn.bAngleMotorSensor THEN
							bJogBackwardsCont := FALSE;
							bInitializeAngle := FALSE;
							iInitializingStep := 1;
						ELSE
							bJogBackwardsCont := TRUE;
						END_IF
						IF fbJog.Error OR bError THEN
							eState := E_StepperState.Error;
						END_IF
					END_IF
				1: bAxisInitialized := TRUE;
					iInitializingStep := 0;
					eState := E_StepperState.Operational;
				
			END_CASE
			
			
			
		E_StepperState.Jog:
			bAxisInitialized := FALSE;
			bAxisReady := FALSE;	
			IF NOT bMovementStarted AND bStepForward THEN
				bJogForward:= TRUE;
				bMovementStarted := TRUE;
				bStepForward := FALSE;
			ELSIF NOT bMovementStarted AND bStepBackward THEN
				bJogBackwards:= TRUE;
				bMovementStarted := TRUE;
				bStepBackward := FALSE;
			END_IF
			IF fbJog.Done THEN
				DoneTmr.IN := TRUE;
				bJogForward:= FALSE;
				bJogBackwards := FALSE;
				bMovementStarted := FALSE;
				eState := E_StepperState.Operational;
			END_IF
			IF fbJog.Error OR fbHalt.Error OR bError THEN
				eState := E_StepperState.Error;
			END_IF
				
				
	E_StepperState.Error:
		fbReset.Execute := FALSE;
		Initialize();
		fbPower.Enable:= FALSE;	
		bError := TRUE;
		IF bResetAxis THEN
			eState := E_StepperState.Offline;
		END_IF
END_CASE


fbPower(
	Axis := fbAxis,
	Enable_Positive := TRUE,
	Enable_Negative := TRUE,
	Status => bAxis1StatusOk,
	Override := 100,
	Error => ,
	ErrorID => nErrorID
	);

fbReset(
	Axis := fbAxis,
	Error =>,
	ErrorID => nErrorID
	);
	
fbJogCont(
	Axis := fbAxis,
	JogForward := bJogForwardCont AND bEstopOk,
	JogBackwards:= bJogBackwardsCont AND bEstopOk,
	Mode := E_JOGMODE.MC_JOGMODE_CONTINOUS,
	Velocity := rStepperVel,
	Acceleration := rStepperAcc, 
	Deceleration := rStepperDec,
	Done =>,
	Error =>,
	ErrorID => nErrorID);
fbMoveAbs(
	Axis := fbAxis,
	Execute := bExecuteMoveAbs AND bEstopOk,
	Position:= rStepCount,
	Velocity := rStepperVel,
	Acceleration := rStepperAcc, 
	Deceleration := rStepperDec,
	Done =>,
	Error =>,
	ErrorID => nErrorID);
fbJog(
	Axis := fbAxis,
	JogForward := bJogForward AND bEstopOk,
	JogBackwards:= bJogBackwards AND bEstopOk,
	Position:= rStepCount,
	Mode := E_JOGMODE.MC_JOGMODE_INCHING,
	Velocity := rStepperVel,
	Acceleration := rStepperAcc, 
	Deceleration := rStepperDec,
	Done =>,
	Error =>,
	ErrorID => nErrorID);

fbHome(
	Axis := fbAxis,
	Execute := bExecuteHoming,
	Position := 0,
	HomingMode := Tc2_MC2.MC_Direct,
	Done => ,
	Error => ,
	ErrorID => nErrorID);

METHOD Initialize : BOOL
VAR_INPUT
END_VAR
bExecuteHoming := FALSE;	
iEncHomingStep := 0;	
bJogForwardCont	:= FALSE;
bJogForward	:= FALSE;	
bMovementStarted := FALSE;		
bJogBackwards := FALSE;
bJogBackwardsCont := FALSE;	
bExecuteMoveAbs := FALSE;
DoneTmr.IN := FALSE;
iInitializingStep := 0;
bExecuteMoveAbs := FALSE;
StopTmr.IN := FALSE;
iEncHomingStep := 0;
bAxisReady	:= FALSE;				
bAxisInitialized := FALSE;
bEnchomingDone := FALSE;
END_METHOD

END_FUNCTION_BLOCK
